FUNCTION FC 105 : VOID
VERSION : 0.1
VAR_TEMP
  Cmd_abbassa_indc : BOOL ;
  Cmd_alza_indc : BOOL ;
  Cmd_abbassa_indc_ibl : BOOL ;
  Cmd_alza_indc_ibl : BOOL ;
  Cmd_sblocca_pezzo : BOOL ;
  Cmd_blocca_pezzo : BOOL ;
  Cmd_sblocca_pezzo_ibl : BOOL ;
  Cmd_blocca_pezzo_ibl : BOOL ;
  Punt1 : DINT ;
  TempoTime : TIME ;
  TempoS5T : S5TIME ;
  Pos_comandata_asse_X : DINT ;
  Pos_comandata_asse_Y : DINT ;
  Tempo_ribaditura : DINT ;
END_VAR
BEGIN
NETWORK
TITLE = ******************       Diagnostica       *******************
NETWORK
TITLE = Allarmi di emergenza
NETWORK
TITLE = Controllo toolcode 
      L     DB106.DBB 0;
      L     W#16#1F;
      AW;
      L     DB110.DBW 36;
      <>I;
      AN    DB110.DBX 78.0;
//      S     "Op10.Bench.Alarms".Emegency.Alarm02
      S     DB104.DBX 9.1;
NETWORK
TITLE = Allarmi di STOP CICLO
NETWORK
TITLE = Controllo anelli adattamento
      A     DB110.DBX 38.0;
      AN    DB106.DBX 0.5;
      O(;
      AN    DB110.DBX 38.0;
      A     DB106.DBX 0.5;
      );
      AN    DB110.DBX 78.1;
      S     DB104.DBX 8.0;
      A     DB110.DBX 38.1;
      AN    DB106.DBX 0.6;
      O(;
      AN    DB110.DBX 38.1;
      A     DB106.DBX 0.6;
      );
      AN    DB110.DBX 78.1;
      S     DB104.DBX 8.1;
NETWORK
TITLE = Allarmi di NON START CICLO
NETWORK
TITLE = Allarmi di Warning
NETWORK
TITLE = Diagnostica: Hold Macchina
      AN    DB100.DBX 2.0;
      A(;
      A     DB100.DBX 0.4;
      AN    DB100.DBX 2.1;
      A     DB105.DBX 10.1;
      O(;
      A     DB100.DBX 0.3;
      A     DB105.DBX 10.0;
      );
      );
      =     DB100.DBX 2.4;
NETWORK
TITLE = ******************          Stati            *******************
      A     DB101.DBX 0.1;
      =     DB105.DBX 10.3;
      A     DB101.DBX 0.2;
      =     DB105.DBX 10.2;
NETWORK
TITLE =
      A     DB55.DBX 10.4;
      =     DB105.DBX 11.3;
      A     DB55.DBX 10.3;
      =     DB105.DBX 11.4;
      A     DB55.DBX 10.2;
      =     DB105.DBX 11.5;
      AN    DB55.DBX 11.2;
      AN    DB55.DBX 12.2;
      =     DB105.DBX 12.4;
NETWORK
TITLE = Stato: Fronte Start Ciclo
      A     DB101.DBX 0.0;
      FP    M 50.2;
      =     DB105.DBX 0.6;
NETWORK
TITLE = Lampade
      A     DB105.DBX 12.2;
      A     DB100.DBX 0.4;
      O     DB105.DBX 0.1;
      =     DB102.DBX 0.0;
      A     DB105.DBX 12.3;
      A     DB100.DBX 0.4;
      O     DB105.DBX 0.1;
      =     DB102.DBX 0.1;
NETWORK
TITLE = Cycle Type
NETWORK
TITLE = ******************         Sistemi           *******************
NETWORK
TITLE = Alza/abbassa Index cassetto
//*************************** COMANDI DA CICLI *************************
      A     DB120.DBX 9.5;
      O     DB120.DBX 12.3;
      O     DB120.DBX 31.7;
      =     DB105.DBX 0.2;
      A     DB120.DBX 10.0;
      A     DB105.DBX 10.2;
      O(;
      A     DB120.DBX 13.0;
      O     DB120.DBX 32.4;
      A     DB105.DBX 10.3;
      );
      =     DB105.DBX 0.3;
//*************************** COMANDI SENZA INTERBLOCCHI ***************
//CMD---------->Comando abbassa index cassetto
//MANUALE
      A     DB70.DBX 12.4;
      A     DB51.DBX 2.3;
      A     DB100.DBX 0.3;
//AUTOMATICO
      O(;
      A     DB100.DBX 0.4;
      AN    DB100.DBX 2.6;
      A     DB105.DBX 0.2;
      );
//SICUREZZA
      A     DB100.DBX 2.4;
      =     #Cmd_abbassa_indc;
//CMD---------->Comando alza index cassetto
//MANUALE
      A     DB70.DBX 12.4;
      A     DB51.DBX 2.2;
      A     DB100.DBX 0.3;
//AUTOMATICO
      O(;
      A     DB100.DBX 0.4;
      AN    DB100.DBX 2.6;
      A     DB105.DBX 0.3;
      );
//SICUREZZA
      A     DB100.DBX 2.4;
      =     #Cmd_alza_indc;
//************************** INTERBLOCCHI (E SEGNALAZIONE) ****************************
      A     DB105.DBX 0.0;
      O     DB105.DBX 10.2;
      O     DB105.DBX 10.3;
      R     DB104.DBX 24.0;
      A     #Cmd_alza_indc;
      A(;
      AN    DB105.DBX 10.2;
      AN    DB105.DBX 10.3;
      );
      S     DB104.DBX 24.0;
// MSG sblocco solo con ribaditrice alta
      A     DB105.DBX 0.0;
      O     DB105.DBX 11.3;
      R     DB104.DBX 24.2;
      A     #Cmd_abbassa_indc;
      AN    DB105.DBX 11.3;
      S     DB104.DBX 24.2;
// MSG sblocco solo con assi fermi
      A     DB105.DBX 0.0;
      O     DB105.DBX 12.4;
      R     DB104.DBX 24.3;
      A     #Cmd_abbassa_indc;
      AN    DB105.DBX 12.4;
      S     DB104.DBX 24.3;
// MSG sblocco solo con pezzo bloccato
      A     DB105.DBX 0.0;
      O     DB105.DBX 10.6;
      R     DB104.DBX 24.4;
      A     #Cmd_abbassa_indc;
      AN    DB105.DBX 10.6;
      S     DB104.DBX 24.4;
//************************** COMANDI CON INTERBLOCCHI ******************************
      AN    DB104.DBX 24.2;
      AN    DB104.DBX 24.3;
      AN    DB104.DBX 24.4;
      A     #Cmd_abbassa_indc;
      =     #Cmd_abbassa_indc_ibl;
      AN    DB104.DBX 24.0;
      A     #Cmd_alza_indc;
      =     #Cmd_alza_indc_ibl;
      CALL  FB 102 , DB 401 (
           DIX 0.0                  := TRUE,
           DIX 0.1                  := #Cmd_alza_indc_ibl,
           DIX 0.2                  := #Cmd_abbassa_indc_ibl,
           DIX 0.3                  := DB101.DBX 0.4,
           DIX 0.4                  := DB101.DBX 0.3,
           DIX 0.5                  := DB105.DBX 0.0,
           DID 2                    := L#2000,
           DIX 6.0                  := FALSE,
           DIX 8.0                  := DB102.DBX 0.3,
           DIX 8.1                  := DB102.DBX 0.2,
           DIX 8.2                  := DB105.DBX 10.5,
           DIX 8.3                  := DB105.DBX 10.4,
           DIX 8.4                  := DB104.DBX 8.2,
           DIX 8.5                  := DB104.DBX 8.3,
           DIX 8.6                  := DB104.DBX 8.4);
NETWORK
TITLE = Blocco/Sblocco pezzo
//*************************** COMANDI DA CICLI *************************
      A     DB120.DBX 13.0;
      O     DB120.DBX 32.4;
      A     DB101.DBX 0.4;
      A     DB105.DBX 10.3;
      =     DB105.DBX 0.4;
      A     DB120.DBX 9.5;
      O     DB120.DBX 10.0;
      =     DB105.DBX 0.5;
//*************************** COMANDI SENZA INTERBLOCCHI ***************
//CMD---------->Comando sblocco
//MANUALE
      A     DB70.DBX 12.5;
      A     DB51.DBX 2.2;
      A     DB100.DBX 0.3;
//AUTOMATICO
      O(;
      A     DB100.DBX 0.4;
      AN    DB100.DBX 2.6;
      A     DB105.DBX 0.4;
      );
//SICUREZZA
      A     DB100.DBX 2.4;
      =     #Cmd_sblocca_pezzo;
//CMD---------->Comando alza ribaditrice
//MANUALE
      A     DB70.DBX 12.5;
      A     DB51.DBX 2.3;
      A     DB100.DBX 0.3;
//AUTOMATICO
      O(;
      A     DB100.DBX 0.4;
      AN    DB100.DBX 2.6;
      A     DB105.DBX 0.5;
      );
//SICUREZZA
      A     DB100.DBX 2.4;
      =     #Cmd_blocca_pezzo;
//************************** INTERBLOCCHI (E SEGNALAZIONE) ****************************
//MSG---> Segnalazione interblocco Movimento ribaditrice non ammesso con motore ribaditrice in marcia
      A     DB105.DBX 0.0;
      O(;
      A     DB105.DBX 10.3;
      A     DB105.DBX 10.5;
      );
      R     DB104.DBX 24.1;
      A     #Cmd_sblocca_pezzo;
      A(;
      AN    DB105.DBX 10.3;
      ON    DB105.DBX 10.5;
      );
      S     DB104.DBX 24.1;
//************************** COMANDI CON INTERBLOCCHI ******************************
//CMD-------------> Comando abbassa e alza
      AN    DB104.DBX 24.1;
      A     #Cmd_sblocca_pezzo;
      =     #Cmd_sblocca_pezzo_ibl;
      A     #Cmd_blocca_pezzo;
      =     #Cmd_blocca_pezzo_ibl;
      CALL  FB 102 , DB 402 (
           DIX 0.0                  := TRUE,
           DIX 0.1                  := #Cmd_sblocca_pezzo_ibl,
           DIX 0.2                  := #Cmd_blocca_pezzo_ibl,
           DIX 0.3                  := DB101.DBX 0.6,
           DIX 0.4                  := DB101.DBX 0.5,
           DIX 0.5                  := DB105.DBX 0.0,
           DID 2                    := L#4000,
           DIX 6.0                  := FALSE,
           DIX 8.0                  := DB102.DBX 0.4,
           DIX 8.1                  := DB102.DBX 0.5,
           DIX 8.2                  := DB105.DBX 10.7,
           DIX 8.3                  := DB105.DBX 10.6,
           DIX 8.4                  := DB104.DBX 8.5,
           DIX 8.5                  := DB104.DBX 8.6,
           DIX 8.6                  := DB104.DBX 8.7);
NETWORK
TITLE = Gestione numero ribaditura in corso
      AN    DB120.DBX 18.0;
      O     DB120.DBX 9.2;
      O     DB120.DBX 10.0;
      O     DB120.DBX 13.0;
      JCN   nAzz;
      L     0;
      T     DB105.DBW 20;
nAzz: NOP   0;
      A     DB120.DBX 10.4;
      FP    M 50.3;
      =     DB105.DBX 11.6;
      AN    DB105.DBX 11.6;
      JC    nIn;
      L     DB105.DBW 20;
      L     1;
      +I;
      T     DB105.DBW 20;
nIn:  NOP   0;
NETWORK
TITLE = Valori posizione ribaditura corrente
      L     DB105.DBW 20;
      L     0;
      >I;
      JC    Cal;
// Punto inesistente
      L     L#0;
      T     DB105.DBD 22;
      T     DB105.DBD 26;
      T     DB105.DBD 30;
      JU    Cen;
Cal:  NOP   0;	// Estrazione dati punto da ricetta
      L     DB105.DBW 20;
      L     1;
      -I;
      ITD;
      L     L#12;
      *D;
      L     L#82;
      +D;
      SLW   3;
      T     #Punt1;
      OPN   DB 110;
      L     DBD [#Punt1];
      T     #Pos_comandata_asse_X;
      L     #Punt1;
      L     32;
      +D;
      T     #Punt1;
      L     DBD [#Punt1];
      T     #Pos_comandata_asse_Y;
      L     #Punt1;
      L     32;
      +D;
      T     #Punt1;
      L     DBD [#Punt1];
      T     #Tempo_ribaditura;
      L     #Pos_comandata_asse_X;
      T     DB105.DBD 22;
      L     #Pos_comandata_asse_Y;
      T     DB105.DBD 26;
      L     #Tempo_ribaditura;
      T     DB105.DBD 30;
Cen:  NOP   0;
NETWORK
TITLE = Impegno, comandi e stati ribaditrice per lavoro su OP10
      A     DB120.DBX 10.0;
      O     DB120.DBX 10.4;
      O     DB120.DBX 11.1;
      O     DB120.DBX 11.6;
      A     DB120.DBX 18.0;
      O(;
      A     DB120.DBX 31.2;
      A     DB120.DBX 40.0;
      );
      =     DB105.DBX 0.7;
      A     DB120.DBX 10.4;
      O     DB120.DBX 11.1;
      O     DB120.DBX 11.6;
      =     DB105.DBX 1.1;
      A     DB120.DBX 11.1;
      A     DB105.DBX 11.0;
      =     DB105.DBX 1.2;
      A     DB120.DBX 9.5;
      AN    DB105.DBX 11.7;
      O     DB120.DBX 11.6;
      O     DB120.DBX 31.2;
      A     DB105.DBX 11.0;
      =     DB105.DBX 1.3;
      A     DB55.DBX 13.0;
      =     DB105.DBX 11.0;
NETWORK
TITLE = Ribaditura
      L     DB105.DBD 30;
      T     #TempoTime;
      CALL  FC 40 (
           $1                       := #TempoTime,
           $2                       := #TempoS5T);
      A     DB120.DBX 11.1;
      A     DB105.DBX 11.5;
      A     DB105.DBX 11.4;
      L     #TempoS5T;
      SD    T 10;
      A     T 10;
      =     DB105.DBX 11.2;
NETWORK
TITLE = Assi - movimenti per lavorazioni OP10
      A     DB120.DBX 10.4;
      A     DB55.DBX 13.0;
      =     DB105.DBX 1.0;
      A     DB55.DBX 11.1;
      A     DB55.DBX 12.1;
      A     DB55.DBX 13.0;
      =     DB105.DBX 11.1;
NETWORK
TITLE = Definizione pezzo buono o scarto
      A     DB120.DBX 12.3;
      S     DB105.DBX 12.2;
      A     DB101.DBX 0.6;
      R     DB105.DBX 12.2;
      A     DB120.DBX 40.0;
      A     DB106.DBX 0.7;
      AN    DB105.DBX 12.2;
      S     DB105.DBX 12.3;
      A     DB101.DBX 0.6;
      R     DB105.DBX 12.3;
END_FUNCTION

FUNCTION FC 106 : VOID
VERSION : 0.1
VAR_INPUT
  ToolType : INT ;
END_VAR
VAR_OUTPUT
  ErrorToolType : BOOL ;
END_VAR
BEGIN
NETWORK
TITLE = Tool 1 - mappa ingressi
// Definizione ingressi E3.0 - E4.6
      L     #ToolType;
      L     1;
      <>I;
      JC    no1;
      SET;
      R     #ErrorToolType;
// Tool 1 - mappa ingressi
      A     I 4.1;
      =     DB106.DBX 0.0;
      A     I 4.2;
      =     DB106.DBX 0.1;
      A     I 4.3;
      =     DB106.DBX 0.2;
      A     I 4.4;
      =     DB106.DBX 0.3;
      A     I 4.5;
      =     DB106.DBX 0.4;
      A     I 4.0;
      =     DB106.DBX 0.5;
      A     I 3.7;
      =     DB106.DBX 0.6;
      A     I 3.6;
      =     DB106.DBX 0.7;
      A     I 3.1;
      =     DB106.DBX 1.0;
      A     I 3.0;
      =     DB106.DBX 1.1;
      A     I 3.3;
      =     DB106.DBX 1.2;
      A     I 3.2;
      =     DB106.DBX 1.3;
      A     I 3.5;
      =     DB106.DBX 1.4;
      A     I 3.4;
      =     DB106.DBX 1.5;
      BEU;
no1:  NOP   0;
NETWORK
TITLE = Tool 2 - mappa ingressi
      L     #ToolType;
      L     2;
      <>I;
      JC    no2;
      SET;
      S     #ErrorToolType;
// Tool 2 - predisposto ma inesistente
      BEU;
no2:  NOP   0;
NETWORK
TITLE = Error Tool Type
      SET;
      S     #ErrorToolType;
END_FUNCTION

FUNCTION FC 120 : VOID
VERSION : 0.1
BEGIN
NETWORK
TITLE =
      A     DB100.DBX 0.4;
      FP    M 50.4;
      =     DB105.DBX 12.0;
      AN    DB100.DBX 2.1;
      AN    DB100.DBX 2.0;
      FP    M 50.5;
      =     DB105.DBX 12.1;
NETWORK
TITLE =
      A     DB105.DBX 12.0;
      O     DB105.DBX 12.1;
      A(;
      AN    DB105.DBX 10.3;
      ON    DB101.DBX 0.4;
      ON    DB101.DBX 0.6;
      );
      S     DB120.DBX 40.0;
      AN    DB100.DBX 0.4;
//      U     "OP10".Diagnostic.Alarm_Stop_Cycle
      O     DB100.DBX 2.0;
      O     DB101.DBX 0.7;
      O     DB120.DBX 37.4;
      R     DB120.DBX 40.0;
      CLR;
      =     DB100.DBX 2.6;
      CALL  FB 121 , DB 431 (
           DIX 0.0                  := DB120.DBX 40.0,
           DIX 0.1                  := DB100.DBX 2.6,
           DIX 0.2                  := FALSE,
           DIX 2.0                  := DB120.DBX 28.0,
           DIX 2.1                  := DB120.DBX 28.1,
           DIX 2.2                  := DB120.DBX 28.2,
           DIW 4                    := DB120.DBW 22,
           DIW 6                    := DB120.DBW 24,
           DIW 8                    := DB120.DBW 26);
NETWORK
TITLE =
      A     DB100.DBX 0.4;
      AN    DB100.DBX 2.1;
      AN    DB100.DBX 2.0;
      AN    DB120.DBX 40.0;
// condizione di sicurezza
      AN    DB101.DBX 0.7;
      =     DB120.DBX 18.0;
      CALL  FB 120 , DB 430 (
           DIX 0.0                  := DB120.DBX 18.0,
           DIX 0.1                  := DB100.DBX 2.6,
           DIX 0.2                  := FALSE,
           DIX 2.0                  := DB120.DBX 6.0,
           DIX 2.1                  := DB120.DBX 6.1,
           DIX 2.2                  := DB120.DBX 6.2,
           DIW 4                    := DB120.DBW 0,
           DIW 6                    := DB120.DBW 2,
           DIW 8                    := DB120.DBW 4);
END_FUNCTION

FUNCTION FC 150 : VOID
VERSION : 0.1
VAR_TEMP
  ErrorToolType : BOOL ;
END_VAR
BEGIN
NETWORK
TITLE =
NETWORK
TITLE =
      CALL  FC 151;
      CALL  FC 156 (
           ToolType                 := DB160.DBW 22,
           ErrorToolType            := #ErrorToolType);
      A     #ErrorToolType;
      A     DB160.DBX 50.0;
//      S     DB154.DBX    0.0
      S     DB154.DBX 8.6;
      CALL  FC 153;
NETWORK
TITLE =
      A     DB55.DBX 0.0;
      =     DB155.DBX 0.0;
      A     DB55.DBX 0.1;
      =     DB155.DBX 0.1;
      A     DB55.DBX 10.1;
      =     DB155.DBX 10.0;
      A     DB55.DBX 10.5;
      =     DB155.DBX 10.1;
      CALL  FC 21 (
           NumDBallarmi             := DB 154,
           Reset_Allarmi            := DB155.DBX 0.0,
           AllarmeEmergenza         := DB150.DBX 2.0,
           AllarmeStopCiclo         := DB150.DBX 2.1,
           AllarmeStartCiclo        := DB150.DBX 2.2,
           AllarmeWarning           := DB150.DBX 2.3);
// Bench mode = Line mode...
      A     DB50.DBX 0.0;
      =     DB150.DBX 0.0;
      A     DB50.DBX 0.1;
      =     DB150.DBX 0.1;
      A     DB50.DBX 0.2;
      =     DB150.DBX 0.2;
      A     DB50.DBX 0.3;
      =     DB150.DBX 0.3;
      A     DB50.DBX 0.4;
      =     DB150.DBX 0.4;
NETWORK
TITLE =
      CALL  FC 155;
      CALL  FC 170;
NETWORK
TITLE =
      CALL  FC 152;
END_FUNCTION

FUNCTION FC 151 : VOID
VERSION : 0.1
VAR_TEMP
  RetVal : WORD ;
  Tastatore : REAL ;
END_VAR
BEGIN
NETWORK
TITLE =
      A     I 10.4;
      =     DB151.DBX 0.2;
      A     I 10.6;
      =     DB151.DBX 0.3;
      A     I 10.5;
      =     DB151.DBX 0.4;
      A     I 10.3;
      =     DB151.DBX 0.5;
      A     I 10.2;
      =     DB151.DBX 0.6;
      A     I 10.1;
      =     DB151.DBX 0.7;
      A     I 10.0;
      =     DB151.DBX 1.0;
NETWORK
TITLE =
      CALL  FC 5 (
           $1                       := P#P 256.0,
           $2                       := L#1088421888,
           $3                       := L#0,
           $4                       := FALSE,
           $5                       := #RetVal,
           $6                       := #Tastatore);
      L     #Tastatore;
      L     DB153.DBD 0;
      -R;
      T     DB151.DBD 6;
END_FUNCTION

FUNCTION FC 152 : VOID
VERSION : 0.1
BEGIN
NETWORK
TITLE =
      A     DB152.DBX 0.0;
      =     Q 0.5;
      A     DB152.DBX 0.1;
      =     Q 0.6;
      A     DB152.DBX 0.2;
      =     Q 2.0;
      A     DB152.DBX 0.3;
      =     Q 2.1;
      A     DB152.DBX 0.4;
      =     Q 1.5;
      A     DB152.DBX 0.5;
      =     Q 1.6;
      A     DB152.DBX 0.6;
      =     Q 1.3;
      A     DB152.DBX 0.7;
      =     Q 1.4;
END_FUNCTION

FUNCTION FC 153 : VOID
VERSION : 0.1
BEGIN
NETWORK
TITLE =
// Impostato da pagina di configurazione su PO
//      L     3.808000e+000
//      T     "Op20.Bench.Config".Offset_Tastatore
END_FUNCTION

FUNCTION FC 155 : VOID
VERSION : 0.1
VAR_TEMP
  Cmd_abbassa_indc : BOOL ;
  Cmd_alza_indc : BOOL ;
  Cmd_abbassa_indc_ibl : BOOL ;
  Cmd_alza_indc_ibl : BOOL ;
  Cmd_sblocca_pezzo : BOOL ;
  Cmd_blocca_pezzo : BOOL ;
  Cmd_sblocca_pezzo_ibl : BOOL ;
  Cmd_blocca_pezzo_ibl : BOOL ;
  Cmd_AlzaGrPiant : BOOL ;
  Cmd_AbbassaGrPiant : BOOL ;
  Cmd_AlzaGrPiant_ibl : BOOL ;
  Cmd_AbbassaGrPiant_ibl : BOOL ;
  Cmd_AlzaPiant : BOOL ;
  Cmd_AbbassaPiant : BOOL ;
  Cmd_AlzaPiant_ibl : BOOL ;
  Cmd_AbbassaPiant_ibl : BOOL ;
  CorsaMinRaggiunta : BOOL ;
  CorsaMaxSuperata : BOOL ;
  TempoTime : TIME ;
  TempoS5T : S5TIME ;
END_VAR
BEGIN
NETWORK
TITLE = ******************       Diagnostica       *******************
NETWORK
TITLE = Allarmi di emergenza
NETWORK
TITLE = Controllo toolcode 
      L     DB156.DBB 0;
      L     W#16#1F;
      AW;
      L     DB160.DBW 24;
      <>I;
      A     DB160.DBX 50.0;
//      S     "Op20.Bench.Alarms".Emegency.Alarm02
      S     DB154.DBX 8.7;
NETWORK
TITLE = Allarmi di STOP CICLO
NETWORK
TITLE = Allarmi di NON START CICLO
NETWORK
TITLE = Allarmi di Warning
NETWORK
TITLE = Diagnostica: Hold Macchina
      AN    DB150.DBX 2.0;
      A(;
      A     DB150.DBX 0.4;
      AN    DB150.DBX 2.1;
      A     DB155.DBX 10.1;
      O(;
      A     DB150.DBX 0.3;
      A     DB155.DBX 10.0;
      );
      );
      =     DB150.DBX 2.4;
NETWORK
TITLE = ******************          Stati            *******************
      AN    DB151.DBX 0.2;
      =     DB155.DBX 10.3;
      A     DB151.DBX 0.2;
      =     DB155.DBX 10.2;
NETWORK
TITLE = Stato: Fronte Start Ciclo
NETWORK
TITLE = Lampade
      A     DB155.DBX 11.3;
      A     DB150.DBX 0.4;
      O     DB155.DBX 0.1;
      =     DB152.DBX 0.0;
      A     DB155.DBX 11.4;
      A     DB150.DBX 0.4;
      O     DB155.DBX 0.1;
      =     DB152.DBX 0.1;
NETWORK
TITLE = Cycle Type
NETWORK
TITLE = ******************         Sistemi           *******************
NETWORK
TITLE = Alza/abbassa Index cassetto
//*************************** COMANDI DA CICLI *************************
      A     DB170.DBX 12.3;
      O     DB170.DBX 31.7;
      =     DB155.DBX 0.2;
      A     DB170.DBX 9.7;
      =     DB155.DBX 0.3;
//*************************** COMANDI SENZA INTERBLOCCHI ***************
//CMD---------->Comando abbassa index cassetto
//MANUALE
      A     DB70.DBX 12.6;
      A     DB51.DBX 2.3;
      A     DB150.DBX 0.3;
//AUTOMATICO
      O(;
      A     DB150.DBX 0.4;
      AN    DB150.DBX 2.6;
      A     DB155.DBX 0.2;
      );
//SICUREZZA
      A     DB150.DBX 2.4;
      =     #Cmd_abbassa_indc;
//CMD---------->Comando alza index cassetto
//MANUALE
      A     DB70.DBX 12.6;
      A     DB51.DBX 2.2;
      A     DB150.DBX 0.3;
//AUTOMATICO
      O(;
      A     DB150.DBX 0.4;
      AN    DB150.DBX 2.6;
      A     DB155.DBX 0.3;
      );
//SICUREZZA
      A     DB150.DBX 2.4;
      =     #Cmd_alza_indc;
//************************** INTERBLOCCHI (E SEGNALAZIONE) ****************************
      A     DB155.DBX 0.0;
      O     DB155.DBX 10.2;
      O     DB155.DBX 10.3;
      R     DB154.DBX 24.0;
      A     #Cmd_alza_indc;
      AN    DB155.DBX 10.2;
      S     DB154.DBX 24.0;
// Msg 
      A     DB155.DBX 0.0;
      O(;
      A     DB155.DBX 10.6;
      A     DB155.DBX 11.0;
      );
      R     DB154.DBX 24.4;
      AN    DB155.DBX 10.6;
      ON    DB155.DBX 11.0;
      A     #Cmd_abbassa_indc;
      S     DB154.DBX 24.4;
//************************** COMANDI CON INTERBLOCCHI ******************************
      AN    DB154.DBX 24.4;
      A     #Cmd_abbassa_indc;
      =     #Cmd_abbassa_indc_ibl;
      AN    DB154.DBX 24.0;
      A     #Cmd_alza_indc;
      =     #Cmd_alza_indc_ibl;
      CALL  FB 102 , DB 403 (
           DIX 0.0                  := TRUE,
           DIX 0.1                  := #Cmd_alza_indc_ibl,
           DIX 0.2                  := #Cmd_abbassa_indc_ibl,
           DIX 0.3                  := DB151.DBX 0.4,
           DIX 0.4                  := DB151.DBX 0.3,
           DIX 0.5                  := DB155.DBX 0.0,
           DID 2                    := L#1500,
           DIX 6.0                  := FALSE,
           DIX 8.0                  := DB152.DBX 0.3,
           DIX 8.1                  := DB152.DBX 0.2,
           DIX 8.2                  := DB155.DBX 10.5,
           DIX 8.3                  := DB155.DBX 10.4,
           DIX 8.4                  := DB154.DBX 8.1,
           DIX 8.5                  := DB154.DBX 8.2,
           DIX 8.6                  := DB154.DBX 8.3);
NETWORK
TITLE = Alza/abbassa gruppo di piantaggio
//*************************** COMANDI DA CICLI *************************
      A     DB170.DBX 11.6;
      O     DB170.DBX 31.2;
      A     DB155.DBX 11.0;
      =     DB155.DBX 0.4;
      A     DB170.DBX 10.4;
      =     DB155.DBX 0.5;
//*************************** COMANDI SENZA INTERBLOCCHI ***************
//CMD---------->Comando alza gruppo
//MANUALE
      A     DB70.DBX 12.7;
      A     DB51.DBX 2.3;
      A     DB150.DBX 0.3;
//AUTOMATICO
      O(;
      A     DB150.DBX 0.4;
      AN    DB150.DBX 2.6;
      A     DB155.DBX 0.4;
      );
//SICUREZZA
//      U     "OP20".Diagnostic.Safe_State
      A     DB155.DBX 10.0;
      =     #Cmd_AlzaGrPiant;
//CMD---------->Comando abbassa gruppo
//MANUALE
      A     DB70.DBX 12.7;
      A     DB51.DBX 2.2;
      A     DB150.DBX 0.3;
//AUTOMATICO
      O(;
      A     DB150.DBX 0.4;
      AN    DB150.DBX 2.6;
      A     DB155.DBX 0.5;
      );
//SICUREZZA
      A     DB150.DBX 2.4;
      =     #Cmd_AbbassaGrPiant;
//************************** INTERBLOCCHI (E SEGNALAZIONE) ****************************
      A     DB155.DBX 0.0;
      O     DB155.DBX 10.2;
      R     DB154.DBX 24.5;
      A     #Cmd_AbbassaGrPiant;
      AN    DB155.DBX 10.2;
      S     DB154.DBX 24.5;
      A     DB155.DBX 0.0;
      O     DB155.DBX 10.5;
      R     DB154.DBX 24.6;
      A     #Cmd_AbbassaGrPiant;
      AN    DB155.DBX 10.5;
      S     DB154.DBX 24.6;
      A     DB155.DBX 0.0;
      O     DB155.DBX 11.0;
      R     DB154.DBX 25.0;
      A     #Cmd_AlzaGrPiant;
      AN    DB155.DBX 11.0;
      S     DB154.DBX 25.0;
//************************** COMANDI CON INTERBLOCCHI ******************************
      AN    DB154.DBX 25.0;
      A     #Cmd_AlzaGrPiant;
      =     #Cmd_AlzaGrPiant_ibl;
      AN    DB154.DBX 24.5;
      AN    DB154.DBX 24.6;
      A     #Cmd_AbbassaGrPiant;
      =     #Cmd_AbbassaGrPiant_ibl;
      CALL  FB 102 , DB 404 (
           DIX 0.0                  := TRUE,
           DIX 0.1                  := #Cmd_AbbassaGrPiant_ibl,
           DIX 0.2                  := #Cmd_AlzaGrPiant_ibl,
           DIX 0.3                  := DB151.DBX 0.7,
           DIX 0.4                  := DB151.DBX 1.0,
           DIX 0.5                  := DB155.DBX 0.0,
           DID 2                    := L#3000,
           DIX 6.0                  := FALSE,
           DIX 8.0                  := DB152.DBX 0.6,
           DIX 8.1                  := DB152.DBX 0.7,
           DIX 8.2                  := DB155.DBX 10.7,
           DIX 8.3                  := DB155.DBX 10.6,
           DIX 8.4                  := DB154.DBX 8.0,
           DIX 8.5                  := DB154.DBX 8.1,
           DIX 8.6                  := DB154.DBX 8.2);
NETWORK
TITLE = Alza/abbassa cilindro di piantaggio
//*************************** COMANDI DA CICLI *************************
      A     DB170.DBX 11.6;
      O     DB170.DBX 31.2;
      =     DB155.DBX 0.6;
      A     DB170.DBX 11.1;
      =     DB155.DBX 0.7;
//*************************** COMANDI SENZA INTERBLOCCHI ***************
//CMD---------->Comando alza gruppo
//MANUALE
      A     DB70.DBX 13.0;
      A     DB51.DBX 2.3;
      A     DB150.DBX 0.3;
//AUTOMATICO
      O(;
      A     DB150.DBX 0.4;
      AN    DB150.DBX 2.6;
      A     DB155.DBX 0.6;
      );
//SICUREZZA
      A     DB150.DBX 2.4;
      =     #Cmd_AlzaPiant;
//CMD---------->Comando abbassa gruppo
//MANUALE
      A     DB70.DBX 13.0;
      A     DB51.DBX 2.2;
      A     DB150.DBX 0.3;
//AUTOMATICO
      O(;
      A     DB150.DBX 0.4;
      AN    DB150.DBX 2.6;
      A     DB155.DBX 0.7;
      );
//SICUREZZA
      A     DB150.DBX 2.4;
      =     #Cmd_AbbassaPiant;
//************************** INTERBLOCCHI (E SEGNALAZIONE) ****************************
      A     #Cmd_AbbassaPiant;
      AN    DB155.DBX 10.2;
      S     DB154.DBX 24.5;
      A     #Cmd_AbbassaPiant;
      AN    DB155.DBX 10.5;
      S     DB154.DBX 24.6;
      A     DB155.DBX 0.0;
      O     DB155.DBX 10.7;
      R     DB154.DBX 24.7;
      A     #Cmd_AbbassaPiant;
      AN    DB155.DBX 10.7;
      S     DB154.DBX 24.7;
//************************** COMANDI CON INTERBLOCCHI ******************************
      A     #Cmd_AlzaPiant;
      =     #Cmd_AlzaPiant_ibl;
      AN    DB154.DBX 24.5;
      AN    DB154.DBX 24.6;
      AN    DB154.DBX 24.7;
      A     #Cmd_AbbassaPiant;
      =     #Cmd_AbbassaPiant_ibl;
      CALL  FB 102 , DB 405 (
           DIX 0.0                  := TRUE,
           DIX 0.1                  := #Cmd_AbbassaPiant_ibl,
           DIX 0.2                  := #Cmd_AlzaPiant_ibl,
           DIX 0.3                  := DB151.DBX 0.5,
           DIX 0.4                  := DB151.DBX 0.6,
           DIX 0.5                  := DB155.DBX 0.0,
           DID 2                    := L#10000,
           DIX 6.0                  := FALSE,
           DIX 8.0                  := DB152.DBX 0.4,
           DIX 8.1                  := DB152.DBX 0.5,
           DIX 8.2                  := DB155.DBX 11.1,
           DIX 8.3                  := DB155.DBX 11.0,
           DIX 8.4                  := DB154.DBX 8.3,
           DIX 8.5                  := DB154.DBX 8.4,
           DIX 8.6                  := DB154.DBX 8.5);
NETWORK
TITLE = Pressatua: controllo ciclo e definizione pezzo OK/KO
      L     DB151.DBD 6;
      L     DB160.DBD 80;
      >=R;
      =     #CorsaMinRaggiunta;
      L     DB151.DBD 6;
      L     DB160.DBD 84;
      >=R;
      =     #CorsaMaxSuperata;
// gestione timeout piantaggio
      L     DB160.DBD 96;
      T     #TempoTime;
      CALL  FC 40 (
           $1                       := #TempoTime,
           $2                       := #TempoS5T);
      A     DB170.DBX 11.1;
      L     #TempoS5T;
      SD    T 21;
// Tempo di piantagio
      L     DB160.DBD 92;
      T     #TempoTime;
      CALL  FC 40 (
           $1                       := #TempoTime,
           $2                       := #TempoS5T);
      A     DB170.DBX 11.1;
      A     #CorsaMinRaggiunta;
      L     #TempoS5T;
      SD    T 22;
// definizione pezzo buono o scartgo
      A     T 21;
      O     #CorsaMaxSuperata;
      A     DB170.DBX 11.1;
      O     DB170.DBX 40.0;
      S     DB155.DBX 11.4;
      A     T 22;
      A     DB170.DBX 11.1;
      S     DB155.DBX 11.3;
      A     DB170.DBX 9.7;
      R     DB155.DBX 11.4;
      R     DB155.DBX 11.3;
// fine operazione di piantaggio
      A     T 22;
      O     T 21;
      A     DB170.DBX 11.1;
      =     DB155.DBX 11.2;
END_FUNCTION

FUNCTION FC 156 : VOID
VERSION : 0.1
VAR_INPUT
  ToolType : INT ;
END_VAR
VAR_OUTPUT
  ErrorToolType : BOOL ;
END_VAR
BEGIN
NETWORK
TITLE = Tool 1 - mappa ingressi
      L     #ToolType;
      L     1;
      <>I;
      JC    no1;
      SET;
      R     #ErrorToolType;
// Tool 1 - mappa ingressi
      A     I 2.3;
      =     DB156.DBX 0.0;
      A     I 2.4;
      =     DB156.DBX 0.1;
      A     I 2.5;
      =     DB156.DBX 0.2;
      A     I 2.6;
      =     DB156.DBX 0.3;
      A     I 2.7;
      =     DB156.DBX 0.4;
      BEU;
no1:  NOP   0;
NETWORK
TITLE = Tool 2 - mappa ingressi
      L     #ToolType;
      L     2;
      <>I;
      JC    no2;
      SET;
      S     #ErrorToolType;
// Tool 2 - predisposto ma inesistente
      BEU;
no2:  NOP   0;
NETWORK
TITLE = Error Tool Type
      SET;
      S     #ErrorToolType;
END_FUNCTION

FUNCTION FC 170 : VOID
VERSION : 0.1
BEGIN
NETWORK
TITLE =
      A     DB150.DBX 0.4;
      FP    M 51.6;
      =     DB155.DBX 11.5;
      AN    DB150.DBX 2.1;
      AN    DB150.DBX 2.0;
      FP    M 51.7;
      =     DB155.DBX 11.6;
NETWORK
TITLE =
      A     DB155.DBX 11.5;
      O     DB155.DBX 11.6;
      A(;
      AN    DB151.DBX 0.3;
      ON    DB151.DBX 1.0;
      ON    DB151.DBX 0.6;
      );
      S     DB170.DBX 40.0;
      AN    DB150.DBX 0.4;
      O     DB150.DBX 2.1;
      O     DB150.DBX 2.0;
      O     DB170.DBX 37.4;
      R     DB170.DBX 40.0;
      CLR;
      =     DB150.DBX 2.6;
      CALL  FB 171 , DB 437 (
           IN_Cm_ON                 := DB170.DBX 40.0,
           IN_HOLD                  := DB150.DBX 2.6,
           IN_STEP                  := FALSE,
           OUT_St_CicloInCorso      := DB170.DBX 28.0,
           OUT_St_CicloTerminatoOK  := DB170.DBX 28.1,
           OUT_St_CicloTerminatoKO  := DB170.DBX 28.2,
           OUT_CicloStato           := DB170.DBW 22,
           OUT_Page                 := DB170.DBW 24,
           OUT_Message              := DB170.DBW 26);
NETWORK
TITLE =
      A     DB150.DBX 0.4;
      AN    DB150.DBX 2.1;
      AN    DB150.DBX 2.0;
      AN    DB170.DBX 40.0;
// condizione di sicurezza
      =     DB170.DBX 18.0;
      CALL  FB 170 , DB 438 (
           IN_Cm_ON                 := DB170.DBX 18.0,
           IN_HOLD                  := DB150.DBX 2.6,
           IN_STEP                  := FALSE,
           OUT_St_CicloInCorso      := DB170.DBX 6.0,
           OUT_St_CicloTerminatoOK  := DB170.DBX 6.1,
           OUT_St_CicloTerminatoKO  := DB170.DBX 6.2,
           OUT_CicloStato           := DB170.DBW 0,
           OUT_Page                 := DB170.DBW 2,
           OUT_Message              := DB170.DBW 4);
END_FUNCTION

FUNCTION FC 200 : VOID
VERSION : 0.1
VAR_TEMP
  ErrorToolType : BOOL ;
END_VAR
BEGIN
NETWORK
TITLE =
NETWORK
TITLE =
      CALL  FC 201;
      CALL  FC 206 (
           ToolType                 := DB210.DBW 34,
           ErrorToolType            := #ErrorToolType);
      A     #ErrorToolType;
      AN    DB210.DBX 78.0;
//      S     DB204.DBX    0.0
      S     DB204.DBX 9.0;
      CALL  FC 203;
NETWORK
TITLE =
      A     DB55.DBX 0.0;
      =     DB205.DBX 0.0;
      A     DB55.DBX 0.1;
      =     DB205.DBX 0.1;
      A     DB55.DBX 10.1;
      =     DB205.DBX 10.0;
      A     DB55.DBX 10.5;
      =     DB205.DBX 10.1;
      CALL  FC 21 (
           NumDBallarmi             := DB 204,
           Reset_Allarmi            := DB205.DBX 0.0,
           AllarmeEmergenza         := DB200.DBX 2.0,
           AllarmeStopCiclo         := DB200.DBX 2.1,
           AllarmeStartCiclo        := DB200.DBX 2.2,
           AllarmeWarning           := DB200.DBX 2.3);
      A     DB50.DBX 0.0;
      =     DB200.DBX 0.0;
      A     DB50.DBX 0.1;
      =     DB200.DBX 0.1;
      A     DB50.DBX 0.2;
      =     DB200.DBX 0.2;
      A     DB50.DBX 0.3;
      =     DB200.DBX 0.3;
      A     DB50.DBX 0.4;
      =     DB200.DBX 0.4;
NETWORK
TITLE =
      CALL  FC 205;
      CALL  FC 220;
NETWORK
TITLE =
      CALL  FC 202;
END_FUNCTION

FUNCTION FC 201 : VOID
VERSION : 0.1
BEGIN
NETWORK
TITLE =
      A     I 6.1;
      =     DB201.DBX 0.0;
      A     I 9.6;
      =     DB201.DBX 0.1;
      AN    I 9.0;
      =     DB201.DBX 0.2;
      A     I 9.1;
      =     DB201.DBX 0.3;
      A     I 9.2;
      =     DB201.DBX 0.4;
      A     I 9.3;
      =     DB201.DBX 0.5;
      A     I 9.4;
      =     DB201.DBX 0.6;
      A     I 9.5;
      =     DB201.DBX 0.7;
      AN    I 1.5;
      =     DB201.DBX 1.0;
END_FUNCTION

FUNCTION FC 202 : VOID
VERSION : 0.1
BEGIN
NETWORK
TITLE =
      A     DB202.DBX 0.0;
      =     Q 0.1;
      A     DB202.DBX 0.1;
      =     Q 0.2;
      A     DB202.DBX 0.2;
      =     Q 2.6;
      A     DB202.DBX 0.3;
      =     Q 2.7;
      A     DB202.DBX 0.4;
      =     Q 3.1;
      A     DB202.DBX 0.5;
      =     Q 3.0;
END_FUNCTION

FUNCTION FC 203 : VOID
VERSION : 0.1
BEGIN
NETWORK
TITLE =
END_FUNCTION

FUNCTION FC 205 : VOID
VERSION : 0.1
VAR_TEMP
  Cmd_abbassa_indc : BOOL ;
  Cmd_alza_indc : BOOL ;
  Cmd_abbassa_indc_ibl : BOOL ;
  Cmd_alza_indc_ibl : BOOL ;
  Cmd_sblocca_pezzo : BOOL ;
  Cmd_blocca_pezzo : BOOL ;
  Cmd_sblocca_pezzo_ibl : BOOL ;
  Cmd_blocca_pezzo_ibl : BOOL ;
  Punt1 : DINT ;
  TempoTime : TIME ;
  TempoS5T : S5TIME ;
  Pos_comandata_asse_X : DINT ;
  Pos_comandata_asse_Y : DINT ;
  Tempo_ribaditura : DINT ;
END_VAR
BEGIN
NETWORK
TITLE = ******************       Diagnostica       *******************
NETWORK
TITLE = Allarmi di emergenza
NETWORK
TITLE = Controllo toolcode 
      L     DB206.DBB 0;
      L     W#16#1F;
      AW;
      L     DB210.DBW 36;
      <>I;
      AN    DB210.DBX 78.0;
//      S     DB204.DBX    0.1
      S     DB204.DBX 9.1;
NETWORK
TITLE = Allarmi di STOP CICLO
NETWORK
TITLE = Controllo anelli adattamento
      A     DB210.DBX 38.0;
      AN    DB206.DBX 0.5;
      O(;
      AN    DB210.DBX 38.0;
      A     DB206.DBX 0.5;
      );
      AN    DB210.DBX 78.1;
      S     DB204.DBX 8.0;
      A     DB210.DBX 38.1;
      AN    DB206.DBX 0.6;
      O(;
      AN    DB210.DBX 38.1;
      A     DB206.DBX 0.6;
      );
      AN    DB210.DBX 78.1;
      S     DB204.DBX 8.1;
NETWORK
TITLE = Allarmi di NON START CICLO
NETWORK
TITLE = Allarmi di Warning
NETWORK
TITLE = Diagnostica: Hold Macchina
      AN    DB200.DBX 2.0;
      A(;
      A     DB200.DBX 0.4;
      AN    DB200.DBX 2.1;
      A     DB205.DBX 10.1;
      O(;
      A     DB200.DBX 0.3;
      A     DB205.DBX 10.0;
      );
      );
      =     DB200.DBX 2.4;
NETWORK
TITLE = ******************          Stati            *******************
      A     DB201.DBX 0.2;
      =     DB205.DBX 10.3;
      A     DB201.DBX 0.3;
      =     DB205.DBX 10.2;
NETWORK
TITLE =
      A     DB55.DBX 10.4;
      =     DB205.DBX 11.3;
      A     DB55.DBX 10.3;
      =     DB205.DBX 11.4;
      A     DB55.DBX 10.2;
      =     DB205.DBX 11.5;
      AN    DB55.DBX 11.2;
      AN    DB55.DBX 12.2;
      =     DB205.DBX 12.4;
NETWORK
TITLE = Stato: Fronte Start Ciclo
      A     DB201.DBX 0.0;
      FP    M 50.7;
      =     DB205.DBX 0.6;
NETWORK
TITLE = Lampade
      A     DB205.DBX 12.2;
      A     DB200.DBX 0.4;
      O     DB205.DBX 0.1;
      =     DB202.DBX 0.0;
      A     DB205.DBX 12.3;
      A     DB200.DBX 0.4;
      O     DB205.DBX 0.1;
      =     DB202.DBX 0.1;
NETWORK
TITLE = Cycle Type
NETWORK
TITLE = ******************         Sistemi           *******************
NETWORK
TITLE = Alza/abbassa Index cassetto
//*************************** COMANDI DA CICLI *************************
      A     DB220.DBX 9.5;
      O     DB220.DBX 12.3;
      O     DB220.DBX 31.7;
      =     DB205.DBX 0.2;
      A     DB220.DBX 10.0;
      A     DB205.DBX 10.2;
      O(;
      A     DB220.DBX 13.0;
      O     DB220.DBX 32.4;
      A     DB205.DBX 10.3;
      );
      =     DB205.DBX 0.3;
//*************************** COMANDI SENZA INTERBLOCCHI ***************
//CMD---------->Comando abbassa index cassetto
//MANUALE
      A     DB70.DBX 13.1;
      A     DB51.DBX 2.3;
      A     DB200.DBX 0.3;
//AUTOMATICO
      O(;
      A     DB200.DBX 0.4;
      AN    DB200.DBX 2.6;
      A     DB205.DBX 0.2;
      );
//SICUREZZA
      A     DB200.DBX 2.4;
      =     #Cmd_abbassa_indc;
//CMD---------->Comando alza index cassetto
//MANUALE
      A     DB70.DBX 13.1;
      A     DB51.DBX 2.2;
      A     DB200.DBX 0.3;
//AUTOMATICO
      O(;
      A     DB200.DBX 0.4;
      AN    DB200.DBX 2.6;
      A     DB205.DBX 0.3;
      );
//SICUREZZA
      A     DB200.DBX 2.4;
      =     #Cmd_alza_indc;
//************************** INTERBLOCCHI (E SEGNALAZIONE) ****************************
      A     DB205.DBX 0.0;
      O     DB205.DBX 10.2;
      O     DB205.DBX 10.3;
      R     DB204.DBX 24.0;
      A     #Cmd_alza_indc;
      A(;
      AN    DB205.DBX 10.2;
      AN    DB205.DBX 10.3;
      );
      S     DB204.DBX 24.0;
// MSG sblocco solo con ribaditrice alta
      A     DB205.DBX 0.0;
      O     DB205.DBX 11.3;
      R     DB204.DBX 24.2;
      A     #Cmd_abbassa_indc;
      AN    DB205.DBX 11.3;
      S     DB204.DBX 24.2;
// MSG sblocco solo con assi fermi
      A     DB205.DBX 0.0;
      O     DB205.DBX 12.4;
      R     DB204.DBX 24.3;
      A     #Cmd_abbassa_indc;
      AN    DB205.DBX 12.4;
      S     DB204.DBX 24.3;
// MSG sblocco solo con pezzo bloccato
      A     DB205.DBX 0.0;
      O     DB205.DBX 10.7;
      R     DB204.DBX 24.4;
      A     #Cmd_abbassa_indc;
      AN    DB205.DBX 10.7;
      S     DB204.DBX 24.4;
//************************** COMANDI CON INTERBLOCCHI ******************************
      AN    DB204.DBX 24.2;
      AN    DB204.DBX 24.3;
      AN    DB204.DBX 24.4;
      A     #Cmd_abbassa_indc;
      =     #Cmd_abbassa_indc_ibl;
      AN    DB204.DBX 24.0;
      A     #Cmd_alza_indc;
      =     #Cmd_alza_indc_ibl;
      CALL  FB 102 , DB 406 (
           DIX 0.0                  := TRUE,
           DIX 0.1                  := #Cmd_alza_indc_ibl,
           DIX 0.2                  := #Cmd_abbassa_indc_ibl,
           DIX 0.3                  := DB201.DBX 0.5,
           DIX 0.4                  := DB201.DBX 0.4,
           DIX 0.5                  := DB205.DBX 0.0,
           DID 2                    := L#3000,
           DIX 6.0                  := FALSE,
           DIX 8.0                  := DB202.DBX 0.3,
           DIX 8.1                  := DB202.DBX 0.2,
           DIX 8.2                  := DB205.DBX 10.5,
           DIX 8.3                  := DB205.DBX 10.4,
           DIX 8.4                  := DB204.DBX 8.2,
           DIX 8.5                  := DB204.DBX 8.3,
           DIX 8.6                  := DB204.DBX 8.4);
NETWORK
TITLE = Blocco/Sblocco pezzo
//*************************** COMANDI DA CICLI *************************
      A     DB220.DBX 9.2;
      O     DB220.DBX 13.0;
      O     DB220.DBX 32.4;
      A     DB201.DBX 0.5;
      A     DB205.DBX 10.3;
      =     DB205.DBX 0.4;
      A     DB220.DBX 9.3;
      O     DB120.DBX 10.0;
      =     DB205.DBX 0.5;
//*************************** COMANDI SENZA INTERBLOCCHI ***************
//CMD---------->Comando sblocco
//MANUALE
      A     DB70.DBX 13.2;
      A     DB51.DBX 2.2;
      A     DB200.DBX 0.3;
//AUTOMATICO
      O(;
      A     DB200.DBX 0.4;
      AN    DB200.DBX 2.6;
      A     DB205.DBX 0.4;
      );
//SICUREZZA
      A     DB200.DBX 2.4;
      =     #Cmd_sblocca_pezzo;
//CMD---------->Comando alza ribaditrice
//MANUALE
      A     DB70.DBX 13.2;
      A     DB51.DBX 2.3;
      A     DB200.DBX 0.3;
//AUTOMATICO
      O(;
      A     DB200.DBX 0.4;
      AN    DB200.DBX 2.6;
      A     DB205.DBX 0.5;
      );
//SICUREZZA
      A     DB200.DBX 2.4;
      =     #Cmd_blocca_pezzo;
//************************** INTERBLOCCHI (E SEGNALAZIONE) ****************************
//MSG---> Segnalazione interblocco Movimento ribaditrice non ammesso con motore ribaditrice in marcia
      A     DB205.DBX 0.0;
      O(;
      A     DB205.DBX 10.3;
      A     DB205.DBX 10.5;
      );
      R     DB204.DBX 24.1;
      A     #Cmd_sblocca_pezzo;
      A(;
      AN    DB205.DBX 10.3;
      ON    DB205.DBX 10.5;
      );
      S     DB204.DBX 24.1;
//************************** COMANDI CON INTERBLOCCHI ******************************
//CMD-------------> Comando abbassa e alza
      AN    DB204.DBX 24.1;
      A     #Cmd_sblocca_pezzo;
      =     #Cmd_sblocca_pezzo_ibl;
      A     #Cmd_blocca_pezzo;
      =     #Cmd_blocca_pezzo_ibl;
      CALL  FB 102 , DB 407 (
           DIX 0.0                  := TRUE,
           DIX 0.1                  := #Cmd_sblocca_pezzo_ibl,
           DIX 0.2                  := #Cmd_blocca_pezzo_ibl,
           DIX 0.3                  := DB201.DBX 0.7,
           DIX 0.4                  := DB201.DBX 0.6,
           DIX 0.5                  := DB205.DBX 0.0,
           DID 2                    := L#3000,
           DIX 6.0                  := FALSE,
           DIX 8.0                  := DB202.DBX 0.4,
           DIX 8.1                  := DB202.DBX 0.5,
           DIX 8.2                  := DB205.DBX 10.6,
           DIX 8.3                  := DB205.DBX 10.7,
           DIX 8.4                  := DB204.DBX 8.5,
           DIX 8.5                  := DB204.DBX 8.6,
           DIX 8.6                  := DB204.DBX 8.7);
NETWORK
TITLE = Gestione numero ribaditura in corso
      AN    DB220.DBX 18.0;
      O     DB220.DBX 9.2;
      O     DB220.DBX 10.0;
      O     DB220.DBX 13.0;
      JCN   nAzz;
      L     0;
      T     DB205.DBW 20;
nAzz: NOP   0;
      A     DB220.DBX 10.4;
      FP    M 50.6;
      =     DB205.DBX 11.6;
      AN    DB205.DBX 11.6;
      JC    nIn;
      L     DB205.DBW 20;
      L     1;
      +I;
      T     DB205.DBW 20;
nIn:  NOP   0;
NETWORK
TITLE = Valori posizione ribaditura corrente
      L     DB205.DBW 20;
      L     0;
      >I;
      JC    Cal;
// Punto inesistente
      L     L#0;
      T     DB205.DBD 22;
      T     DB205.DBD 26;
      T     DB205.DBD 30;
      JU    Cen;
Cal:  NOP   0;	// Estrazione dati punto da ricetta
      L     DB205.DBW 20;
      DEC   1;
      ITD;
      L     L#12;
      *D;
      L     L#82;
      +D;
      SLW   3;
      T     #Punt1;
      OPN   DB 210;
      L     DBD [#Punt1];
      T     #Pos_comandata_asse_X;
      L     #Punt1;
      L     32;
      +D;
      T     #Punt1;
      L     DBD [#Punt1];
      T     #Pos_comandata_asse_Y;
      L     #Punt1;
      L     32;
      +D;
      T     #Punt1;
      L     DBD [#Punt1];
      T     #Tempo_ribaditura;
      L     #Pos_comandata_asse_X;
      T     DB205.DBD 22;
      L     #Pos_comandata_asse_Y;
      T     DB205.DBD 26;
      L     #Tempo_ribaditura;
      T     DB205.DBD 30;
Cen:  NOP   0;
NETWORK
TITLE = Impegno, comandi e stati ribaditrice per lavoro su OP10
      A     DB220.DBX 10.0;
      O     DB220.DBX 10.4;
      O     DB220.DBX 11.1;
      O     DB220.DBX 11.6;
      A     DB220.DBX 18.0;
      O(;
      A     DB220.DBX 31.2;
      A     DB220.DBX 40.0;
      );
      =     DB205.DBX 0.7;
      A     DB220.DBX 10.4;
      O     DB220.DBX 11.1;
      O     DB220.DBX 11.6;
      =     DB205.DBX 1.1;
      A     DB220.DBX 11.1;
      A     DB205.DBX 11.0;
      =     DB205.DBX 1.2;
      A     DB220.DBX 9.5;
      AN    DB205.DBX 11.7;
      O     DB220.DBX 11.6;
      O     DB220.DBX 31.2;
      A     DB205.DBX 11.0;
      =     DB205.DBX 1.3;
      A     DB55.DBX 13.1;
      =     DB205.DBX 11.0;
NETWORK
TITLE = Ribaditura
      L     DB205.DBD 30;
      T     #TempoTime;
      CALL  FC 40 (
           $1                       := #TempoTime,
           $2                       := #TempoS5T);
      A     DB220.DBX 11.1;
      A     DB205.DBX 11.5;
      A     DB205.DBX 11.4;
      L     #TempoS5T;
      SD    T 11;
      A     T 11;
      =     DB205.DBX 11.2;
NETWORK
TITLE = Assi - movimenti per lavorazioni OP10
      A     DB220.DBX 10.4;
      A     DB55.DBX 13.1;
      =     DB205.DBX 1.0;
      A     DB55.DBX 11.1;
      A     DB55.DBX 12.1;
      A     DB55.DBX 13.1;
      =     DB205.DBX 11.1;
NETWORK
TITLE = Definizione pezzo buono o scarto
      A     DB220.DBX 12.3;
      S     DB205.DBX 12.2;
      A     DB201.DBX 0.7;
      R     DB205.DBX 12.2;
      A     DB220.DBX 40.0;
      A     DB206.DBX 0.7;
      AN    DB205.DBX 12.2;
      S     DB205.DBX 12.3;
      A     DB201.DBX 0.7;
      R     DB205.DBX 12.3;
END_FUNCTION

FUNCTION FC 206 : VOID
VERSION : 0.1
VAR_INPUT
  ToolType : INT ;
END_VAR
VAR_OUTPUT
  ErrorToolType : BOOL ;
END_VAR
BEGIN
NETWORK
TITLE = Tool 1 - mappa ingressi
      L     #ToolType;
      L     1;
      <>I;
      JC    no1;
      SET;
      R     #ErrorToolType;
// Tool 1 - mappa ingressi
      A     I 7.0;
      =     DB206.DBX 0.0;
      A     I 7.1;
      =     DB206.DBX 0.1;
      A     I 7.2;
      =     DB206.DBX 0.2;
      A     I 7.3;
      =     DB206.DBX 0.3;
      A     I 7.4;
      =     DB206.DBX 0.4;
      A     I 5.1;
      =     DB206.DBX 0.5;
      A     I 5.2;
      =     DB206.DBX 0.6;
      A     I 5.0;
      =     DB206.DBX 0.7;
      BEU;
no1:  NOP   0;
NETWORK
TITLE = Tool 2 - mappa ingressi
      L     #ToolType;
      L     2;
      <>I;
      JC    no2;
      SET;
      S     #ErrorToolType;
// Tool 2 - predisposto ma inesistente
      BEU;
no2:  NOP   0;
NETWORK
TITLE = Error Tool Type
      SET;
      S     #ErrorToolType;
END_FUNCTION

FUNCTION FC 220 : VOID
VERSION : 0.1
BEGIN
NETWORK
TITLE =
      A     DB200.DBX 0.4;
      FP    M 51.0;
      =     DB205.DBX 12.0;
      AN    DB200.DBX 2.1;
      AN    DB200.DBX 2.0;
      FP    M 51.1;
      =     DB205.DBX 12.1;
NETWORK
TITLE =
      A     DB205.DBX 12.0;
      O     DB205.DBX 12.1;
      A(;
      AN    DB205.DBX 10.3;
      ON    DB201.DBX 0.5;
      ON    DB201.DBX 0.7;
      );
      S     DB220.DBX 40.0;
      AN    DB200.DBX 0.4;
      O     DB200.DBX 2.1;
      O     DB200.DBX 2.0;
      O     DB201.DBX 1.0;
      O     DB220.DBX 37.4;
      R     DB220.DBX 40.0;
      CLR;
      =     DB200.DBX 2.6;
      CALL  FB 221 , DB 435 (
           DIX 0.0                  := DB220.DBX 40.0,
           DIX 0.1                  := DB200.DBX 2.6,
           DIX 0.2                  := FALSE,
           DIX 2.0                  := DB220.DBX 28.0,
           DIX 2.1                  := DB220.DBX 28.1,
           DIX 2.2                  := DB220.DBX 28.2,
           DIW 4                    := DB220.DBW 22,
           DIW 6                    := DB220.DBW 24,
           DIW 8                    := DB220.DBW 26);
NETWORK
TITLE =
      A     DB200.DBX 0.4;
      AN    DB200.DBX 2.1;
      AN    DB200.DBX 2.0;
      AN    DB220.DBX 40.0;
// condizione di sicurezza
      AN    DB201.DBX 1.0;
      =     DB220.DBX 18.0;
      CALL  FB 220 , DB 436 (
           DIX 0.0                  := DB220.DBX 18.0,
           DIX 0.1                  := DB200.DBX 2.6,
           DIX 0.2                  := FALSE,
           DIX 2.0                  := DB220.DBX 6.0,
           DIX 2.1                  := DB220.DBX 6.1,
           DIX 2.2                  := DB220.DBX 6.2,
           DIW 4                    := DB220.DBW 0,
           DIW 6                    := DB220.DBW 2,
           DIW 8                    := DB220.DBW 4);
END_FUNCTION

DATA_BLOCK DB 50
VERSION : 0.1
UDT 250
BEGIN
END_DATA_BLOCK

DATA_BLOCK DB 51
VERSION : 0.1
  STRUCT
   Q_Ribaditrice : BOOL ;
   Q_protezione_uscite : BOOL ;
   Q_Protez_circ_emergena : BOOL ;	//161QF1
   Q_Automatici_230_V : BOOL ;	//162F1-162F2-162F3-162F4
   Aux_OK : BOOL ;
   Ripari_OK : BOOL ;
   Anomalia_Condizionatore : BOOL ;
   Sequenza_fasi_OK : BOOL ;
   PLC_OK : BOOL ;	//Feedback relè PLC ok
   Chiave_Blocc_Porta_SX : BOOL ;
   Chiave_Blocc_Porta_DX : BOOL ;
   P_TestLampade : BOOL ;
   P_StartCiclo : BOOL ;	//??? che fa ???
   P_StopCiclo : BOOL ;
   S_Manuale : BOOL ;
   S_Automatico : BOOL ;
   Q_Azionam_Asse_X : BOOL ;
   Q_Azionam_Asse_Y : BOOL ;
   Jog_piu : BOOL ;
   Jog_meno : BOOL ;
   P_reset_allarmi : BOOL ;
   Pressostato_aria : BOOL ;
   Ribaditrice_bassa : BOOL ;
   Ribaditrice_alta : BOOL ;
   Press_aria_dpoop_EMG : BOOL ;
   Extracorsa_X : BOOL ;
   Extracorsa_Y : BOOL ;
   Ris_33 : BOOL ;
   Ris_34 : BOOL ;
   Ris_35 : BOOL ;
   Ris_36 : BOOL ;
   Ris_37 : BOOL ;
  END_STRUCT ;	
BEGIN
   Q_Ribaditrice := TRUE;
   Q_protezione_uscite := TRUE;
   Q_Protez_circ_emergena := TRUE;
   Q_Automatici_230_V := TRUE;
   Aux_OK := TRUE;
   Ripari_OK := TRUE;
   Sequenza_fasi_OK := TRUE;
   PLC_OK := TRUE;
   Chiave_Blocc_Porta_SX := TRUE;
   Chiave_Blocc_Porta_DX := TRUE;
   S_Automatico := TRUE;
   Q_Azionam_Asse_X := TRUE;
   Q_Azionam_Asse_Y := TRUE;
   Pressostato_aria := TRUE;
   Ribaditrice_alta := TRUE;
   Press_aria_dpoop_EMG := TRUE;
END_DATA_BLOCK

DATA_BLOCK DB 52
VERSION : 0.1
  STRUCT
   PLC_OK : BOOL ;
   Valvola_generale_aria : BOOL ;	//TOLTO!!!
   Marcia_ribaditrice : BOOL ;
   EV_abbassa_ribaditrice : BOOL ;
   Spare_0_4 : BOOL ;
   Blocco_porta_SX : BOOL ;
   Blocco_porta_DX : BOOL ;
   Lampeggiante_allarmi : BOOL ;
   LampPorteChiuse : BOOL ;
  END_STRUCT ;	
BEGIN
   PLC_OK := TRUE;
   Blocco_porta_SX := TRUE;
   Blocco_porta_DX := TRUE;
   LampPorteChiuse := TRUE;
END_DATA_BLOCK

DATA_BLOCK DB 53
VERSION : 0.1
  STRUCT
   Vel_max_assi_auto : DINT ;	//
   Vel_max_assi_man : DINT ;
   Accel_assi_auto : DINT ;
   Accel_assi_man : DINT ;
   Offset_attrezzo_OP10_X : DINT ;	//
   Offset_attrezzo_OP10_Y : DINT ;
   Offset_attrezzo_OP40_X : DINT ;	//
   Offset_attrezzo_OP40_Y : DINT ;
  END_STRUCT ;	
BEGIN
   Vel_max_assi_auto := L#15000;
   Vel_max_assi_man := L#15000;
   Accel_assi_auto := L#100;
   Accel_assi_man := L#100;
   Offset_attrezzo_OP10_X := L#71501;
   Offset_attrezzo_OP10_Y := L#47116;
   Offset_attrezzo_OP40_X := L#371523;
   Offset_attrezzo_OP40_Y := L#47047;
END_DATA_BLOCK

DATA_BLOCK DB 54
VERSION : 0.1
  STRUCT
   Emegency : STRUCT
    Alarm01 : BOOL ;	//Q_protezione_uscite
    Alarm02 : BOOL ;	//Protez_circ_emergena
    Alarm03 : BOOL ;	//Sequenza_fasi_OK
    Alarm04 : BOOL ;	//Q_Azionam_Asse_X
    Alarm05 : BOOL ;	//Q_Azionam_Asse_Y
    Alarm06 : BOOL ;	//Manca aria
    Alarm07 : BOOL ;	//Valvola aria inceppata
    Alarm08 : BOOL ;	//Errore comunicazione con Azionamento asse X
    Alarm09 : BOOL ;	//Errore comunicazione con Azionamento asse Y
    Alarm10 : BOOL ;	//Errore comunicazione con CU Azionamento asse X
    Alarm11 : BOOL ;	//Errore comunicazione con CU Azionamento asse Y
    Alarm12 : BOOL ;	//Extracorsa asse X
    Alarm13 : BOOL ;	//Extracorsa asse Y
    Alarm14 : BOOL ;	//Errore Relè PLC OK
    Alarm15 : BOOL ;
    Alarm16 : BOOL ;
    Alarm17 : BOOL ;
    Alarm18 : BOOL ;
    Alarm19 : BOOL ;
    Alarm20 : BOOL ;
    Alarm21 : BOOL ;
    Alarm22 : BOOL ;
    Alarm23 : BOOL ;
    Alarm24 : BOOL ;
    Alarm25 : BOOL ;
    Alarm26 : BOOL ;
    Alarm27 : BOOL ;
    Alarm28 : BOOL ;
    Alarm29 : BOOL ;
    Alarm30 : BOOL ;
    Alarm31 : BOOL ;
    Alarm32 : BOOL ;
    Alarm33 : BOOL ;
    Alarm34 : BOOL ;
    Alarm35 : BOOL ;
    Alarm36 : BOOL ;
    Alarm37 : BOOL ;
    Alarm38 : BOOL ;
    Alarm39 : BOOL ;
    Alarm40 : BOOL ;
    Alarm41 : BOOL ;
    Alarm42 : BOOL ;
    Alarm43 : BOOL ;
    Alarm44 : BOOL ;
    Alarm45 : BOOL ;
    Alarm46 : BOOL ;
    Alarm47 : BOOL ;
    Alarm48 : BOOL ;
    Alarm49 : BOOL ;
    Alarm50 : BOOL ;
    Alarm51 : BOOL ;
    Alarm52 : BOOL ;
    Alarm53 : BOOL ;
    Alarm54 : BOOL ;
    Alarm55 : BOOL ;
    Alarm56 : BOOL ;
    Alarm57 : BOOL ;
    Alarm58 : BOOL ;
    Alarm59 : BOOL ;
    Alarm60 : BOOL ;
    Alarm61 : BOOL ;
    Alarm62 : BOOL ;
    Alarm63 : BOOL ;
    Alarm64 : BOOL ;
   END_STRUCT ;
   StopCycle : STRUCT
    Alarm01 : BOOL ;	//Ribaditrice non bassa
    Alarm02 : BOOL ;	//Ribaditrice non alta
    Alarm03 : BOOL ;	//Incongruenza sensori ribaditrice
    Alarm04 : BOOL ;	//Porte non chiuse
    Alarm05 : BOOL ;	//Chiave non Bloccata Porta SX
    Alarm06 : BOOL ;	//Chiave non Bloccata Porta DX
    Alarm07 : BOOL ;	//asse X bloccato con Ribaditrice non alta
    Alarm08 : BOOL ;	//asse Y bloccato con Ribaditrice non alta
    Alarm09 : BOOL ;
    Alarm10 : BOOL ;
    Alarm11 : BOOL ;	//Macchina in emergenza
    Alarm12 : BOOL ;
    Alarm13 : BOOL ;
    Alarm14 : BOOL ;
    Alarm15 : BOOL ;
    Alarm16 : BOOL ;
    Alarm17 : BOOL ;
    Alarm18 : BOOL ;
    Alarm19 : BOOL ;
    Alarm20 : BOOL ;
    Alarm21 : BOOL ;
    Alarm22 : BOOL ;
    Alarm23 : BOOL ;
    Alarm24 : BOOL ;
    Alarm25 : BOOL ;
    Alarm26 : BOOL ;
    Alarm27 : BOOL ;
    Alarm28 : BOOL ;
    Alarm29 : BOOL ;
    Alarm30 : BOOL ;
    Alarm31 : BOOL ;
    Alarm32 : BOOL ;
    Alarm33 : BOOL ;
    Alarm34 : BOOL ;
    Alarm35 : BOOL ;
    Alarm36 : BOOL ;
    Alarm37 : BOOL ;
    Alarm38 : BOOL ;
    Alarm39 : BOOL ;
    Alarm40 : BOOL ;
    Alarm41 : BOOL ;
    Alarm42 : BOOL ;
    Alarm43 : BOOL ;
    Alarm44 : BOOL ;
    Alarm45 : BOOL ;
    Alarm46 : BOOL ;
    Alarm47 : BOOL ;
    Alarm48 : BOOL ;
    Alarm49 : BOOL ;
    Alarm50 : BOOL ;
    Alarm51 : BOOL ;
    Alarm52 : BOOL ;
    Alarm53 : BOOL ;
    Alarm54 : BOOL ;
    Alarm55 : BOOL ;
    Alarm56 : BOOL ;
    Alarm57 : BOOL ;
    Alarm58 : BOOL ;
    Alarm59 : BOOL ;
    Alarm60 : BOOL ;
    Alarm61 : BOOL ;
    Alarm62 : BOOL ;
    Alarm63 : BOOL ;
    Alarm64 : BOOL ;
   END_STRUCT ;
   RestartCycle : STRUCT
    Alarm01 : BOOL ;
    Alarm02 : BOOL ;
    Alarm03 : BOOL ;
    Alarm04 : BOOL ;
    Alarm05 : BOOL ;
    Alarm06 : BOOL ;
    Alarm07 : BOOL ;
    Alarm08 : BOOL ;
    Alarm09 : BOOL ;
    Alarm10 : BOOL ;
    Alarm11 : BOOL ;
    Alarm12 : BOOL ;
    Alarm13 : BOOL ;
    Alarm14 : BOOL ;
    Alarm15 : BOOL ;
    Alarm16 : BOOL ;
    Alarm17 : BOOL ;
    Alarm18 : BOOL ;
    Alarm19 : BOOL ;
    Alarm20 : BOOL ;
    Alarm21 : BOOL ;
    Alarm22 : BOOL ;
    Alarm23 : BOOL ;
    Alarm24 : BOOL ;
    Alarm25 : BOOL ;
    Alarm26 : BOOL ;
    Alarm27 : BOOL ;
    Alarm28 : BOOL ;
    Alarm29 : BOOL ;
    Alarm30 : BOOL ;
    Alarm31 : BOOL ;
    Alarm32 : BOOL ;
    Alarm33 : BOOL ;
    Alarm34 : BOOL ;
    Alarm35 : BOOL ;
    Alarm36 : BOOL ;
    Alarm37 : BOOL ;
    Alarm38 : BOOL ;
    Alarm39 : BOOL ;
    Alarm40 : BOOL ;
    Alarm41 : BOOL ;
    Alarm42 : BOOL ;
    Alarm43 : BOOL ;
    Alarm44 : BOOL ;
    Alarm45 : BOOL ;
    Alarm46 : BOOL ;
    Alarm47 : BOOL ;
    Alarm48 : BOOL ;
    Alarm49 : BOOL ;
    Alarm50 : BOOL ;
    Alarm51 : BOOL ;
    Alarm52 : BOOL ;
    Alarm53 : BOOL ;
    Alarm54 : BOOL ;
    Alarm55 : BOOL ;
    Alarm56 : BOOL ;
    Alarm57 : BOOL ;
    Alarm58 : BOOL ;
    Alarm59 : BOOL ;
    Alarm60 : BOOL ;
    Alarm61 : BOOL ;
    Alarm62 : BOOL ;
    Alarm63 : BOOL ;
    Alarm64 : BOOL ;
   END_STRUCT ;
   Warning : STRUCT
    Alarm01 : BOOL ;	//Q_Ribaditrice
    Alarm02 : BOOL ;	//Q_Automatici_230_V
    Alarm03 : BOOL ;	//Anomalia_Condizionatore
    Alarm04 : BOOL ;	//Ribaditrice bloccata con motore ribaditrice ferma
    Alarm05 : BOOL ;	//Marcia ribaditrice solo con cassetti OP10 e OP40 indexati
    Alarm06 : BOOL ;	//Dicesa dibaditrice solo con cassetti OP10 e OP40 indexati
    Alarm07 : BOOL ;	//Marcia assi solo con cassetti OP10 e OP40 indexati
    Alarm08 : BOOL ;
    Alarm09 : BOOL ;
    Alarm10 : BOOL ;
    Alarm11 : BOOL ;
    Alarm12 : BOOL ;
    Alarm13 : BOOL ;
    Alarm14 : BOOL ;
    Alarm15 : BOOL ;
    Alarm16 : BOOL ;
    Alarm17 : BOOL ;
    Alarm18 : BOOL ;
    Alarm19 : BOOL ;
    Alarm20 : BOOL ;
    Alarm21 : BOOL ;
    Alarm22 : BOOL ;
    Alarm23 : BOOL ;
    Alarm24 : BOOL ;
    Alarm25 : BOOL ;
    Alarm26 : BOOL ;
    Alarm27 : BOOL ;
    Alarm28 : BOOL ;
    Alarm29 : BOOL ;
    Alarm30 : BOOL ;
    Alarm31 : BOOL ;
    Alarm32 : BOOL ;
    Alarm33 : BOOL ;
    Alarm34 : BOOL ;
    Alarm35 : BOOL ;
    Alarm36 : BOOL ;
    Alarm37 : BOOL ;
    Alarm38 : BOOL ;
    Alarm39 : BOOL ;
    Alarm40 : BOOL ;
    Alarm41 : BOOL ;
    Alarm42 : BOOL ;
    Alarm43 : BOOL ;
    Alarm44 : BOOL ;
    Alarm45 : BOOL ;
    Alarm46 : BOOL ;
    Alarm47 : BOOL ;
    Alarm48 : BOOL ;
    Alarm49 : BOOL ;
    Alarm50 : BOOL ;
    Alarm51 : BOOL ;
    Alarm52 : BOOL ;
    Alarm53 : BOOL ;
    Alarm54 : BOOL ;
    Alarm55 : BOOL ;
    Alarm56 : BOOL ;
    Alarm57 : BOOL ;
    Alarm58 : BOOL ;
    Alarm59 : BOOL ;
    Alarm60 : BOOL ;
    Alarm61 : BOOL ;
    Alarm62 : BOOL ;
    Alarm63 : BOOL ;
    Alarm64 : BOOL ;
   END_STRUCT ;
  END_STRUCT ;	
BEGIN
END_DATA_BLOCK

DATA_BLOCK DB 55
VERSION : 0.1
  STRUCT
   Command : STRUCT 	//
    Reset_allarmi : BOOL ;
    TestLampade : BOOL ;	//da programmare sul pannello operatore
    Abbassa_ribaditrice : BOOL ;
    Alza_ribaditrice : BOOL ;
    Marcia_ribaditrice : BOOL ;	//manca ingresso
    Marcia_manuale_ribaditr : BOOL ;
    Posiziona_Assi : BOOL ;
    ris_0_7 : BOOL ;
    AsseX_Enable : BOOL ;
    AsseX_StartPosizionam : BOOL ;
    AsseX_ris_2 : BOOL ;
    AsseX_ris_3 : BOOL ;
    AsseX_ris_4 : BOOL ;
    AsseX_ris_5 : BOOL ;
    AsseX_ris_6 : BOOL ;
    AsseX_ris_7 : BOOL ;
    AsseY_Enable : BOOL ;
    AsseY_StartPosizionam : BOOL ;
    AsseY_ris_2 : BOOL ;
    AsseY_ris_3 : BOOL ;
    AsseY_ris_4 : BOOL ;
    AsseY_ris_5 : BOOL ;
    AsseY_ris_6 : BOOL ;
    AsseY_ris_7 : BOOL ;
    PrenotaRib_OP10 : BOOL ;
    PrenotaRib_OP40 : BOOL ;
    ris_w4 : WORD ;
    ris_w6 : DWORD ;
   END_STRUCT ;
   State : STRUCT 	//da ind. 10
    PLC_OK : BOOL ;
    Porte_chiuse : BOOL ;
    Ribadit_Motore_in_marcia : BOOL ;
    Ribaditrice_bassa : BOOL ;
    Ribaditrice_alta : BOOL ;
    Porte_chiuse_e_bloccate : BOOL ;
    Cassetto_OP10_indexato : BOOL ;
    Cassetto_OP40_indexato : BOOL ;
    AsseX_referenziato : BOOL ;
    AsseX_posizioneRaggiunta : BOOL ;
    AsseX_inMovimento : BOOL ;
    Ris_1_3 : BOOL ;
    AsseX_ExtracorsaOK : BOOL ;
    AsseX_FC_indietro : BOOL ;
    AsseX_FC_avanti : BOOL ;
    AsseX_Pronto : BOOL ;
    AsseY_referenziato : BOOL ;
    AsseY_posizioneRaggiunta : BOOL ;
    AsseY_inMovimento : BOOL ;
    Ris_2_3 : BOOL ;
    AsseY_ExtracorsaOK : BOOL ;
    AsseY_FC_indietro : BOOL ;
    AsseY_FC_avanti : BOOL ;
    AsseY_pronto : BOOL ;
    Ribad_prenotata_da_OP10 : BOOL ;
    Ribad_prenotata_da_OP40 : BOOL ;
    FP_IngressoInPag_TeachIn : BOOL ;
    FP_NumPuntoCambiato : BOOL ;
    FP_RichiestaLeggiPunto : BOOL ;
    FP_RichiestaSalvaPunto : BOOL ;
    FP_RichiestaTeachInPunto : BOOL ;
    ris_w4 : WORD ;
    ris_w6 : DWORD ;
   END_STRUCT ;
   Data : STRUCT 	//da ind. 20
    ris_X_0 : INT ;
    AsseX_Accelerazione : INT ;
    AsseX_Decellerazione : INT ;
    AsseX_Velocita : DINT ;
    AsseX_PosizioneComandata : DINT ;
    AsseX_PosizioneAttuale : DINT ;
    AsseX_CodiceErrore : BYTE ;
    AsseX_ris20 : WORD ;
    AsseX_ris22 : DWORD ;
    AsseX_ris26 : DWORD ;
    ris_Y_30 : INT ;
    AsseY_Accelerazione : INT ;
    AsseY_Decellerazione : INT ;
    AsseY_Velocita : DINT ;
    AsseY_PosizioneComandata : DINT ;
    AsseY_PosizioneAttuale : DINT ;
    AsseY_CodiceErrore : BYTE ;
    AsseY_ris50 : WORD ;
    AsseY_ris52 : DWORD ;
    AsseY_ris56 : DWORD ;
    PuntoInTeachIn : INT ;
    ris_82 : INT ;
    ris_84 : INT ;
    ris_86 : DINT ;
    ris_90 : ARRAY  [0 .. 40 ] OF INT ;
   END_STRUCT ;
  END_STRUCT ;	
BEGIN
   Command.AsseX_Enable := TRUE;
   Command.AsseY_Enable := TRUE;
   State.PLC_OK := TRUE;
   State.Porte_chiuse := TRUE;
   State.Ribaditrice_alta := TRUE;
   State.Porte_chiuse_e_bloccate := TRUE;
   State.Cassetto_OP10_indexato := TRUE;
   State.Cassetto_OP40_indexato := TRUE;
   State.AsseX_referenziato := TRUE;
   State.AsseX_ExtracorsaOK := TRUE;
   State.AsseX_Pronto := TRUE;
   State.AsseY_referenziato := TRUE;
   State.AsseY_ExtracorsaOK := TRUE;
   State.AsseY_pronto := TRUE;
   Data.AsseX_Accelerazione := 100;
   Data.AsseX_Decellerazione := 100;
   Data.AsseX_Velocita := L#15000;
   Data.AsseX_PosizioneAttuale := L#347483;
   Data.AsseY_Accelerazione := 100;
   Data.AsseY_Decellerazione := 100;
   Data.AsseY_Velocita := L#15000;
   Data.AsseY_PosizioneAttuale := L#23007;
   Data.PuntoInTeachIn := 1;
END_DATA_BLOCK

DATA_BLOCK DB 60
VERSION : 0.1
  STRUCT
   Coord_Ribaditrice : UDT 200;
  END_STRUCT ;	
BEGIN
// 22 bytes; values not shown
END_DATA_BLOCK

DATA_BLOCK DB 70
VERSION : 0.1
  STRUCT
   OP_System_Data : STRUCT
    PageDisplayed : INT ;
    Year_Byte0 : BYTE ;
    Year_Byte1 : BYTE ;
    Month_byte0 : BYTE ;
    Month_byte1 : BYTE ;
    Day_byte0 : BYTE ;
    Day_byte1 : BYTE ;
    HH : BYTE ;
    MM : BYTE ;
    NewPage : INT ;
   END_STRUCT ;
   Commands : STRUCT 	//da indirizzo 12
    Man_Alza_Abb_Ribaditrice : BOOL ;
    Man_Marcia_Ribaditrice : BOOL ;
    Man_Jog_AsseX : BOOL ;
    Man_Jog_AsseY : BOOL ;
    Man_10_IndexCassetto : BOOL ;
    Man_10_BloccoPezzo : BOOL ;
    Man_20_IndexCassetto : BOOL ;
    Man_20_GruppoPiantaggio : BOOL ;
    Man_20_Piantaggio : BOOL ;
    Man_40_IndexCassetto : BOOL ;
    Man_40_BloccoPezzo : BOOL ;
    Man_disp_2_3 : BOOL ;
    Man_disp_2_4 : BOOL ;
    Man_disp_2_5 : BOOL ;
    Man_disp_2_6 : BOOL ;
    Man_disp_2_7 : BOOL ;
    Man_VaiAlPunto : WORD ;
    Reset_Allarmi : BOOL ;
    Cmd_VaiAlPunto : BOOL ;
    Cmd_TeachInPunto : BOOL ;
    Cmd_SalvaPunto : BOOL ;
    Cmd_LeggiPunto : BOOL ;
    Ris_16_5 : BOOL ;
    ris_w18 : DINT ;
    ris_w22 : DINT ;
   END_STRUCT ;
   States : STRUCT 	//da indirizzo 26
    RibaditriceAlta : BOOL ;
    RibaditriceBassa : BOOL ;
    RibaditriceFerma : BOOL ;
    RibaditriceInMarcia : BOOL ;
    OP10IndexCassSbloccato : BOOL ;
    OP10IndexCassBloccato : BOOL ;
    OP10PezzoSbloccato : BOOL ;
    OP10PezzoBloccato : BOOL ;
    AsseXIndietro : BOOL ;
    AsseXAvanti : BOOL ;
    AsseYIndietro : BOOL ;
    AsseYAvanti : BOOL ;
    OP20IndexCassSbloccato : BOOL ;
    OP20IndexCassBloccato : BOOL ;
    OP20GrPiantaggioAlto : BOOL ;
    OP20GrPiantaggioBasso : BOOL ;
    OP20PiantaggioAlto : BOOL ;
    OP20PiantaggioBasso : BOOL ;
    OP40IndexCassSbloccato : BOOL ;
    OP40IndexCassBloccato : BOOL ;
    OP40PezzoSbloccato : BOOL ;
    OP40PezzoBloccato : BOOL ;
    ris_w30 : INT ;
    ris_w32 : DINT ;
   END_STRUCT ;
   Data : STRUCT 	//da indirizzo 36
    AsseX_PosizioneAttuale : DINT ;	//Valori assoluti assi
    AsseY_PosizioneAttuale : DINT ;	//Valori assoluti assi
    PosizionePunzone : REAL ;
    Cmd_Override_man : INT ;
    Cmd_Override_auto : INT ;
    AsseX_PosAttualeOP10 : DINT ;
    AsseY_PosAttualeOP10 : DINT ;
    AsseX_PosAttualeOP40 : DINT ;
    AsseY_PosAttualeOP40 : DINT ;
    Cmd_PuntoSelezionato : INT ;
    Min_PerSelezionePunto : INT ;
    Max_PerSelezionePunto : INT ;
    X_PosPuntoSelezionato : DINT ;
    Y_PosPuntoSelezionato : DINT ;
    TempoRibad_PuntoSelez : DINT ;
    ris_array : ARRAY  [0 .. 15 ] OF REAL ;
   END_STRUCT ;
   cycles : STRUCT 	//indirizzo 150
    OP10_cycle_general : BOOL ;
    OP10_cycle_restore : BOOL ;
    OP20_cycle_general : BOOL ;
    OP20_cycle_restore : BOOL ;
    OP40_cycle_general : BOOL ;
    OP40_cycle_restore : BOOL ;
    OP10_message : INT ;
    OP10_spacer : INT ;
    OP40_message : INT ;
    OP40_spacer : INT ;
    OP20_message : INT ;
    Line_State : INT ;
    ris_w8 : INT ;
    ris_array : ARRAY  [0 .. 16 ] OF INT ;
   END_STRUCT ;
  END_STRUCT ;	
BEGIN
   OP_System_Data.PageDisplayed := 120;
   OP_System_Data.Year_Byte1 := B#16#10;
   OP_System_Data.Month_byte1 := B#16#4;
   OP_System_Data.Day_byte1 := B#16#6;
   OP_System_Data.HH := B#16#21;
   OP_System_Data.MM := B#16#39;
   OP_System_Data.NewPage := 120;
   Commands.Man_Marcia_Ribaditrice := TRUE;
   States.RibaditriceAlta := TRUE;
   States.RibaditriceFerma := TRUE;
   States.OP10IndexCassBloccato := TRUE;
   States.OP10PezzoBloccato := TRUE;
   States.OP20IndexCassSbloccato := TRUE;
   States.OP20GrPiantaggioAlto := TRUE;
   States.OP20PiantaggioAlto := TRUE;
   States.OP40IndexCassBloccato := TRUE;
   States.OP40PezzoSbloccato := TRUE;
   Data.AsseX_PosizioneAttuale := L#347483;
   Data.AsseY_PosizioneAttuale := L#23007;
   Data.PosizionePunzone := -3.808000e+00;
   Data.Cmd_Override_man := 100;
   Data.Cmd_Override_auto := 40;
   Data.AsseX_PosAttualeOP10 := L#275982;
   Data.AsseY_PosAttualeOP10 := L#-24109;
   Data.AsseX_PosAttualeOP40 := L#-24040;
   Data.AsseY_PosAttualeOP40 := L#-24040;
   Data.Cmd_PuntoSelezionato := 1;
   Data.Min_PerSelezionePunto := 1;
   Data.Max_PerSelezionePunto := 1;
   Data.X_PosPuntoSelezionato := L#-24040;
   Data.Y_PosPuntoSelezionato := L#-24040;
   Data.TempoRibad_PuntoSelez := L#3000;
   cycles.OP10_cycle_general := TRUE;
   cycles.OP20_cycle_general := TRUE;
   cycles.OP40_cycle_general := TRUE;
   cycles.OP10_message := 2;
   cycles.OP40_message := 4;
   cycles.OP20_message := 2;
   cycles.Line_State := 4;
END_DATA_BLOCK

DATA_BLOCK DB 100
VERSION : 0.1
UDT 250
BEGIN
END_DATA_BLOCK

DATA_BLOCK DB 101
VERSION : 0.1
  STRUCT
   P_Consenso_operatore : BOOL ;	//(start ciclo)
   Cassetto_fuori : BOOL ;
   Cassetto_dentro : BOOL ;
   Index_cassetto_Giu : BOOL ;
   Index_cassetto_Su : BOOL ;
   Sblocco_pezzo_Giu : BOOL ;
   Sblocco_pezzo_Su : BOOL ;
   PulStopCiclo : BOOL ;
  END_STRUCT ;	
BEGIN
   Cassetto_fuori := TRUE;
   Index_cassetto_Su := TRUE;
   Sblocco_pezzo_Su := TRUE;
END_DATA_BLOCK

DATA_BLOCK DB 102
VERSION : 0.1
  STRUCT
   Fine_ciclo_OK : BOOL ;	//
   Fine_ciclo_NON_OK : BOOL ;
   EV_abb_index_cassetto : BOOL ;
   EV_alza_index_cassetto : BOOL ;
   EV_sblocco_pezzo : BOOL ;
   EV_blocco_pezzo : BOOL ;	//??? esiste?
  END_STRUCT ;	
BEGIN
   EV_alza_index_cassetto := TRUE;
   EV_sblocco_pezzo := TRUE;
END_DATA_BLOCK

DATA_BLOCK DB 103
VERSION : 0.1
  STRUCT
   dummy : INT ;
  END_STRUCT ;	
BEGIN
END_DATA_BLOCK

DATA_BLOCK DB 104
VERSION : 0.1
  STRUCT
   Emegency : STRUCT
    Alarm01 : BOOL ;	//OP10 ToolType error
    Alarm02 : BOOL ;	//OP10 ToolCode error
    Alarm03 : BOOL ;
    Alarm04 : BOOL ;
    Alarm05 : BOOL ;
    Alarm06 : BOOL ;
    Alarm07 : BOOL ;
    Alarm08 : BOOL ;
    Alarm09 : BOOL ;	//
    Alarm10 : BOOL ;	//
    Alarm11 : BOOL ;	//
    Alarm12 : BOOL ;	//
    Alarm13 : BOOL ;	//
    Alarm14 : BOOL ;	//
    Alarm15 : BOOL ;
    Alarm16 : BOOL ;
    Alarm17 : BOOL ;
    Alarm18 : BOOL ;
    Alarm19 : BOOL ;
    Alarm20 : BOOL ;
    Alarm21 : BOOL ;
    Alarm22 : BOOL ;
    Alarm23 : BOOL ;
    Alarm24 : BOOL ;
    Alarm25 : BOOL ;
    Alarm26 : BOOL ;
    Alarm27 : BOOL ;
    Alarm28 : BOOL ;
    Alarm29 : BOOL ;
    Alarm30 : BOOL ;
    Alarm31 : BOOL ;
    Alarm32 : BOOL ;
    Alarm33 : BOOL ;
    Alarm34 : BOOL ;
    Alarm35 : BOOL ;
    Alarm36 : BOOL ;
    Alarm37 : BOOL ;
    Alarm38 : BOOL ;
    Alarm39 : BOOL ;
    Alarm40 : BOOL ;
    Alarm41 : BOOL ;
    Alarm42 : BOOL ;
    Alarm43 : BOOL ;
    Alarm44 : BOOL ;
    Alarm45 : BOOL ;
    Alarm46 : BOOL ;
    Alarm47 : BOOL ;
    Alarm48 : BOOL ;
    Alarm49 : BOOL ;
    Alarm50 : BOOL ;
    Alarm51 : BOOL ;
    Alarm52 : BOOL ;
    Alarm53 : BOOL ;
    Alarm54 : BOOL ;
    Alarm55 : BOOL ;
    Alarm56 : BOOL ;
    Alarm57 : BOOL ;
    Alarm58 : BOOL ;
    Alarm59 : BOOL ;
    Alarm60 : BOOL ;
    Alarm61 : BOOL ;
    Alarm62 : BOOL ;
    Alarm63 : BOOL ;
    Alarm64 : BOOL ;
   END_STRUCT ;
   StopCycle : STRUCT
    Alarm01 : BOOL ;	//Errore rilevamento anello di adattamento 1
    Alarm02 : BOOL ;	//Errore rilevamento anello di adattamento 2
    Alarm03 : BOOL ;	//Index cassetto non alto
    Alarm04 : BOOL ;	//Index cassetto non basso
    Alarm05 : BOOL ;	//Incongruenza sensori index cassetto
    Alarm06 : BOOL ;	//Cilindro sblocco pezzo non avanti
    Alarm07 : BOOL ;	//Cilindro sblocco pezzo non indietro
    Alarm08 : BOOL ;	//Incongruenza sensori cilindro sblocco pezzo
    Alarm09 : BOOL ;	//OP10 ToolType error
    Alarm10 : BOOL ;	//OP10 ToolCode error
    Alarm11 : BOOL ;
    Alarm12 : BOOL ;
    Alarm13 : BOOL ;
    Alarm14 : BOOL ;
    Alarm15 : BOOL ;
    Alarm16 : BOOL ;
    Alarm17 : BOOL ;
    Alarm18 : BOOL ;
    Alarm19 : BOOL ;
    Alarm20 : BOOL ;
    Alarm21 : BOOL ;
    Alarm22 : BOOL ;
    Alarm23 : BOOL ;
    Alarm24 : BOOL ;
    Alarm25 : BOOL ;
    Alarm26 : BOOL ;
    Alarm27 : BOOL ;
    Alarm28 : BOOL ;
    Alarm29 : BOOL ;
    Alarm30 : BOOL ;
    Alarm31 : BOOL ;
    Alarm32 : BOOL ;
    Alarm33 : BOOL ;
    Alarm34 : BOOL ;
    Alarm35 : BOOL ;
    Alarm36 : BOOL ;
    Alarm37 : BOOL ;
    Alarm38 : BOOL ;
    Alarm39 : BOOL ;
    Alarm40 : BOOL ;
    Alarm41 : BOOL ;
    Alarm42 : BOOL ;
    Alarm43 : BOOL ;
    Alarm44 : BOOL ;
    Alarm45 : BOOL ;
    Alarm46 : BOOL ;
    Alarm47 : BOOL ;
    Alarm48 : BOOL ;
    Alarm49 : BOOL ;
    Alarm50 : BOOL ;
    Alarm51 : BOOL ;
    Alarm52 : BOOL ;
    Alarm53 : BOOL ;
    Alarm54 : BOOL ;
    Alarm55 : BOOL ;
    Alarm56 : BOOL ;
    Alarm57 : BOOL ;
    Alarm58 : BOOL ;
    Alarm59 : BOOL ;
    Alarm60 : BOOL ;
    Alarm61 : BOOL ;
    Alarm62 : BOOL ;
    Alarm63 : BOOL ;
    Alarm64 : BOOL ;
   END_STRUCT ;
   RestartCycle : STRUCT
    Alarm01 : BOOL ;
    Alarm02 : BOOL ;
    Alarm03 : BOOL ;
    Alarm04 : BOOL ;
    Alarm05 : BOOL ;
    Alarm06 : BOOL ;
    Alarm07 : BOOL ;
    Alarm08 : BOOL ;
    Alarm09 : BOOL ;
    Alarm10 : BOOL ;
    Alarm11 : BOOL ;
    Alarm12 : BOOL ;
    Alarm13 : BOOL ;
    Alarm14 : BOOL ;
    Alarm15 : BOOL ;
    Alarm16 : BOOL ;
    Alarm17 : BOOL ;
    Alarm18 : BOOL ;
    Alarm19 : BOOL ;
    Alarm20 : BOOL ;
    Alarm21 : BOOL ;
    Alarm22 : BOOL ;
    Alarm23 : BOOL ;
    Alarm24 : BOOL ;
    Alarm25 : BOOL ;
    Alarm26 : BOOL ;
    Alarm27 : BOOL ;
    Alarm28 : BOOL ;
    Alarm29 : BOOL ;
    Alarm30 : BOOL ;
    Alarm31 : BOOL ;
    Alarm32 : BOOL ;
    Alarm33 : BOOL ;
    Alarm34 : BOOL ;
    Alarm35 : BOOL ;
    Alarm36 : BOOL ;
    Alarm37 : BOOL ;
    Alarm38 : BOOL ;
    Alarm39 : BOOL ;
    Alarm40 : BOOL ;
    Alarm41 : BOOL ;
    Alarm42 : BOOL ;
    Alarm43 : BOOL ;
    Alarm44 : BOOL ;
    Alarm45 : BOOL ;
    Alarm46 : BOOL ;
    Alarm47 : BOOL ;
    Alarm48 : BOOL ;
    Alarm49 : BOOL ;
    Alarm50 : BOOL ;
    Alarm51 : BOOL ;
    Alarm52 : BOOL ;
    Alarm53 : BOOL ;
    Alarm54 : BOOL ;
    Alarm55 : BOOL ;
    Alarm56 : BOOL ;
    Alarm57 : BOOL ;
    Alarm58 : BOOL ;
    Alarm59 : BOOL ;
    Alarm60 : BOOL ;
    Alarm61 : BOOL ;
    Alarm62 : BOOL ;
    Alarm63 : BOOL ;
    Alarm64 : BOOL ;
   END_STRUCT ;
   Warning : STRUCT
    Alarm01 : BOOL ;	//Blocco movimento index cassetto se cassetto non dentro o non fuori
    Alarm02 : BOOL ;	//Blocco sblocco pezzo se cassetto non fuori
    Alarm03 : BOOL ;	//Sblocco index solo con ribaditrice alta
    Alarm04 : BOOL ;	//Sblocco index solo con assi fermi
    Alarm05 : BOOL ;	//Sblocco index solo pezzo bloccato
    Alarm06 : BOOL ;
    Alarm07 : BOOL ;
    Alarm08 : BOOL ;
    Alarm09 : BOOL ;
    Alarm10 : BOOL ;
    Alarm11 : BOOL ;
    Alarm12 : BOOL ;
    Alarm13 : BOOL ;
    Alarm14 : BOOL ;
    Alarm15 : BOOL ;
    Alarm16 : BOOL ;
    Alarm17 : BOOL ;
    Alarm18 : BOOL ;
    Alarm19 : BOOL ;
    Alarm20 : BOOL ;
    Alarm21 : BOOL ;
    Alarm22 : BOOL ;
    Alarm23 : BOOL ;
    Alarm24 : BOOL ;
    Alarm25 : BOOL ;
    Alarm26 : BOOL ;
    Alarm27 : BOOL ;
    Alarm28 : BOOL ;
    Alarm29 : BOOL ;
    Alarm30 : BOOL ;
    Alarm31 : BOOL ;
    Alarm32 : BOOL ;
    Alarm33 : BOOL ;
    Alarm34 : BOOL ;
    Alarm35 : BOOL ;
    Alarm36 : BOOL ;
    Alarm37 : BOOL ;
    Alarm38 : BOOL ;
    Alarm39 : BOOL ;
    Alarm40 : BOOL ;
    Alarm41 : BOOL ;
    Alarm42 : BOOL ;
    Alarm43 : BOOL ;
    Alarm44 : BOOL ;
    Alarm45 : BOOL ;
    Alarm46 : BOOL ;
    Alarm47 : BOOL ;
    Alarm48 : BOOL ;
    Alarm49 : BOOL ;
    Alarm50 : BOOL ;
    Alarm51 : BOOL ;
    Alarm52 : BOOL ;
    Alarm53 : BOOL ;
    Alarm54 : BOOL ;
    Alarm55 : BOOL ;
    Alarm56 : BOOL ;
    Alarm57 : BOOL ;
    Alarm58 : BOOL ;
    Alarm59 : BOOL ;
    Alarm60 : BOOL ;
    Alarm61 : BOOL ;
    Alarm62 : BOOL ;
    Alarm63 : BOOL ;
    Alarm64 : BOOL ;
   END_STRUCT ;
  END_STRUCT ;	
BEGIN
   Warning.Alarm05 := TRUE;
END_DATA_BLOCK

DATA_BLOCK DB 105
VERSION : 0.1
  STRUCT
   Command : STRUCT 	//
    Reset_allarmi : BOOL ;
    TestLampade : BOOL ;
    Abbassa_index_cassetto : BOOL ;
    Alza_index_cassetto : BOOL ;
    Sblocca_pezzo : BOOL ;
    Blocca_pezzo : BOOL ;
    FP_Consenso_operatore : BOOL ;
    Prenota_ribaditrice : BOOL ;
    Vai_in_posizione_assi : BOOL ;
    Marcia_ribaditrice : BOOL ;
    Abbassa_ribaditrice : BOOL ;
    Alza_ribaditrice : BOOL ;
    ris_w2 : DWORD ;
    ris_w6 : DWORD ;
   END_STRUCT ;
   State : STRUCT
    Porte_chiuse : BOOL ;
    Porte_chiuse_e_bloccate : BOOL ;
    Cassetto_dentro : BOOL ;
    Cassetto_fuori : BOOL ;
    Index_cassetto_basso : BOOL ;
    Index_cassetto_alto : BOOL ;
    Pezzo_sbloccato : BOOL ;
    Pezzo_bloccato : BOOL ;
    _Ribaditrice_a_disposiz : BOOL ;
    _Assi_posiz_raggiunta : BOOL ;
    Ribaditura_effettuata : BOOL ;
    Ribaditrice_alta : BOOL ;
    Ribaditrice_bassa : BOOL ;
    Ribaditrice_in_marcia : BOOL ;
    FP_stato_20_generale : BOOL ;
    _Ribad_in_fuori_ingombro : BOOL ;
    FP_Mode_automatic : BOOL ;
    FP_uscita_da_allarme : BOOL ;
    Ribaditura_pezzo_OK : BOOL ;
    Ribaditura_pezzo_KO : BOOL ;
    Assi_fermi : BOOL ;
    ris_w4 : WORD ;
    ris_w6 : DWORD ;
   END_STRUCT ;
   Data : STRUCT
    Num_punto_in_lavorazione : INT ;
    Pos_comandata_asse_X : DINT ;	//Punto in lavorazione
    Pos_comandata_asse_Y : DINT ;	//Punto in lavorazione
    Tempo_ribaditura : DINT ;	//Punto in lavorazione
    ris_w2 : DWORD ;
    ris_w6 : DWORD ;
   END_STRUCT ;
  END_STRUCT ;	
BEGIN
   State.Porte_chiuse := TRUE;
   State.Porte_chiuse_e_bloccate := TRUE;
   State.Cassetto_fuori := TRUE;
   State.Index_cassetto_alto := TRUE;
   State.Pezzo_bloccato := TRUE;
   State.Ribaditrice_alta := TRUE;
   State.Assi_fermi := TRUE;
END_DATA_BLOCK

DATA_BLOCK DB 106
VERSION : 0.1
  STRUCT
   ToolCode_Bit_0 : BOOL ;	//
   ToolCode_Bit_1 : BOOL ;
   ToolCode_Bit_2 : BOOL ;
   ToolCode_Bit_3 : BOOL ;
   ToolCode_Bit_4 : BOOL ;
   Anello_1_Inserito : BOOL ;
   Anello_2_Inserito : BOOL ;
   Presenza_nozzle_ring : BOOL ;
   Spacer_1_presente : BOOL ;
   Spacer_1_invertito : BOOL ;
   Spacer_2_presente : BOOL ;
   Spacer_2_invertito : BOOL ;
   Spacer_3_presente : BOOL ;
   Spacer_3_invertito : BOOL ;
   Ris_1_6 : BOOL ;
   Ris_1_7 : BOOL ;
  END_STRUCT ;	
BEGIN
   ToolCode_Bit_1 := TRUE;
   Anello_1_Inserito := TRUE;
END_DATA_BLOCK

DATA_BLOCK DB 108
VERSION : 0.1
  STRUCT
   DB_VAR : INT ;	//Variabile jolly provvisoria
  END_STRUCT ;	
BEGIN
END_DATA_BLOCK

DATA_BLOCK DB 110
VERSION : 0.1
  STRUCT
   ID_Ricetta : INT ;
   PartNumber : ARRAY  [0 .. 31 ] OF //Part number in lavorazione
   CHAR ;
   ToolType : INT ;	//Tool type
   ToolCode : INT ;	//Codice su attrezzo - ingressi digitali
   Anello1Abilitato : BOOL ;
   Anello2Abilitato : BOOL ;
   Velocita_asse_X : DINT ;
   Velocita_asse_Y : DINT ;
   spare48 : DINT ;
   spare52 : DINT ;
   spare56 : DINT ;
   spare60 : DINT ;
   spare64 : DINT ;
   spare68 : DINT ;
   spare72 : DINT ;
   spare76 : INT ;
   Disable : STRUCT 	//da indirizzo 78
    CkCodicePortapezzo : BOOL ;
    CkPresAnelloAdattamento : BOOL ;
    CkPresenzaNozzleRing : BOOL ;
    CkPresenzaSpacer1 : BOOL ;
    CkPresenzaSpacer2 : BOOL ;
    CkPresenzaSpacer3 : BOOL ;
    CheckSpare1 : BOOL ;
    CheckSpare2 : BOOL ;
    CheckSpare3 : BOOL ;
    CheckSpare4 : BOOL ;
   END_STRUCT ;
   NumeroPosizioni : INT ;
   posizioni : ARRAY  [0 .. 19 ] OF //da indirizzo 82
   STRUCT
    X : DINT ;	//1/100 mm
    Y : DINT ;	//1/100 mm
    TempoRibaditura : DINT ;	//msec
   END_STRUCT ;
   spare : ARRAY  [0 .. 38 ] OF INT ;
  END_STRUCT ;	
BEGIN
   ID_Ricetta := 1;
   PartNumber[0] := 'R';
   PartNumber[1] := 'P';
   PartNumber[2] := 'V';
   PartNumber[3] := 'O';
   PartNumber[4] := ' ';
   PartNumber[5] := 'A';
   PartNumber[6] := 'P';
   PartNumber[7] := 'O';
   PartNumber[8] := '0';
   PartNumber[9] := '1';
   PartNumber[10] := ' ';
   PartNumber[11] := ' ';
   PartNumber[12] := ' ';
   PartNumber[13] := ' ';
   PartNumber[14] := ' ';
   PartNumber[15] := ' ';
   PartNumber[16] := ' ';
   PartNumber[17] := ' ';
   PartNumber[18] := ' ';
   PartNumber[19] := ' ';
   PartNumber[20] := ' ';
   PartNumber[21] := ' ';
   PartNumber[22] := ' ';
   PartNumber[23] := ' ';
   PartNumber[24] := ' ';
   PartNumber[25] := ' ';
   PartNumber[26] := ' ';
   PartNumber[27] := ' ';
   PartNumber[28] := ' ';
   PartNumber[29] := ' ';
   PartNumber[30] := ' ';
   PartNumber[31] := ' ';
   ToolType := 1;
   ToolCode := 2;
   Anello1Abilitato := TRUE;
   Velocita_asse_X := L#100000;
   Velocita_asse_Y := L#100000;
   NumeroPosizioni := 3;
   posizioni[0].X := L#-24040;
   posizioni[0].Y := L#-24040;
   posizioni[0].TempoRibaditura := L#3000;
   posizioni[1].X := L#-15440;
   posizioni[1].Y := L#30290;
   posizioni[1].TempoRibaditura := L#3000;
   posizioni[2].X := L#33580;
   posizioni[2].Y := L#5320;
   posizioni[2].TempoRibaditura := L#3000;
END_DATA_BLOCK

DATA_BLOCK DB 120
VERSION : 0.1
  STRUCT
   General : UDT 200;
   Restore : UDT 200;
  END_STRUCT ;	
BEGIN
// 44 bytes; values not shown
END_DATA_BLOCK

DATA_BLOCK DB 150
VERSION : 0.1
UDT 250
BEGIN
END_DATA_BLOCK

DATA_BLOCK DB 151
VERSION : 0.1
  STRUCT
   Ris_0_0 : BOOL ;
   Ris_0_1 : BOOL ;
   Cassetto_dentro : BOOL ;	//manca ingresso
   Index_cassetto_Giu : BOOL ;	//manca ingresso
   Index_cassetto_Su : BOOL ;	//manca ingresso
   Piantaggio_Giu : BOOL ;
   Piantaggio_Su : BOOL ;
   Gruppo_piantaggio_Giu : BOOL ;
   Gruppo_piantaggio_Su : BOOL ;
   Ris_w2 : WORD ;
   ris_w3 : WORD ;
   _Posizione_Punzone : REAL ;	//mm
  END_STRUCT ;	
BEGIN
   Cassetto_dentro := TRUE;
   Index_cassetto_Giu := TRUE;
   Piantaggio_Su := TRUE;
   Gruppo_piantaggio_Su := TRUE;
   _Posizione_Punzone := -3.808000e+00;
END_DATA_BLOCK

DATA_BLOCK DB 152
VERSION : 0.1
  STRUCT
   Fine_ciclo_OK : BOOL ;	//
   Fine_ciclo_NON_OK : BOOL ;
   EV_abb_index_cassetto : BOOL ;	//Libera index cassetto su zona piantaggio
   EV_alza_index_cassetto : BOOL ;	//Blocca index cassetto su zona piantaggio
   EV_abbassa_piantaggio : BOOL ;
   EV_alza_piantaggio : BOOL ;
   EV_abb_grupp_piantaggio : BOOL ;
   EV_alz_grupp_piantaggio : BOOL ;
  END_STRUCT ;	
BEGIN
   Fine_ciclo_OK := TRUE;
   EV_abb_index_cassetto := TRUE;
   EV_alza_piantaggio := TRUE;
   EV_alz_grupp_piantaggio := TRUE;
END_DATA_BLOCK

DATA_BLOCK DB 153
VERSION : 0.1
  STRUCT
   Offset_Tastatore : REAL ;	//
  END_STRUCT ;	
BEGIN
   Offset_Tastatore := 3.808000e+00;
END_DATA_BLOCK

DATA_BLOCK DB 154
VERSION : 0.1
  STRUCT
   Emegency : STRUCT
    Alarm01 : BOOL ;	//OP20 ToolType error
    Alarm02 : BOOL ;	//OP20 ToolCode error
    Alarm03 : BOOL ;
    Alarm04 : BOOL ;
    Alarm05 : BOOL ;
    Alarm06 : BOOL ;
    Alarm07 : BOOL ;
    Alarm08 : BOOL ;
    Alarm09 : BOOL ;	//
    Alarm10 : BOOL ;	//
    Alarm11 : BOOL ;	//
    Alarm12 : BOOL ;	//
    Alarm13 : BOOL ;	//
    Alarm14 : BOOL ;	//
    Alarm15 : BOOL ;
    Alarm16 : BOOL ;
    Alarm17 : BOOL ;
    Alarm18 : BOOL ;
    Alarm19 : BOOL ;
    Alarm20 : BOOL ;
    Alarm21 : BOOL ;
    Alarm22 : BOOL ;
    Alarm23 : BOOL ;
    Alarm24 : BOOL ;
    Alarm25 : BOOL ;
    Alarm26 : BOOL ;
    Alarm27 : BOOL ;
    Alarm28 : BOOL ;
    Alarm29 : BOOL ;
    Alarm30 : BOOL ;
    Alarm31 : BOOL ;
    Alarm32 : BOOL ;
    Alarm33 : BOOL ;
    Alarm34 : BOOL ;
    Alarm35 : BOOL ;
    Alarm36 : BOOL ;
    Alarm37 : BOOL ;
    Alarm38 : BOOL ;
    Alarm39 : BOOL ;
    Alarm40 : BOOL ;
    Alarm41 : BOOL ;
    Alarm42 : BOOL ;
    Alarm43 : BOOL ;
    Alarm44 : BOOL ;
    Alarm45 : BOOL ;
    Alarm46 : BOOL ;
    Alarm47 : BOOL ;
    Alarm48 : BOOL ;
    Alarm49 : BOOL ;
    Alarm50 : BOOL ;
    Alarm51 : BOOL ;
    Alarm52 : BOOL ;
    Alarm53 : BOOL ;
    Alarm54 : BOOL ;
    Alarm55 : BOOL ;
    Alarm56 : BOOL ;
    Alarm57 : BOOL ;
    Alarm58 : BOOL ;
    Alarm59 : BOOL ;
    Alarm60 : BOOL ;
    Alarm61 : BOOL ;
    Alarm62 : BOOL ;
    Alarm63 : BOOL ;
    Alarm64 : BOOL ;
   END_STRUCT ;
   StopCycle : STRUCT
    Alarm01 : BOOL ;	//Gruppo di piantaggio non basso
    Alarm02 : BOOL ;	//Gruppo di piantaggio non alto
    Alarm03 : BOOL ;	//Incongruenza sensori gruppo di piantaggio
    Alarm04 : BOOL ;	//piantaggio non basso
    Alarm05 : BOOL ;	//piantaggio non alto
    Alarm06 : BOOL ;	//Incongruenza sensori piantaggio
    Alarm07 : BOOL ;	//OP20 ToolType error
    Alarm08 : BOOL ;	//OP20 ToolCode error
    Alarm09 : BOOL ;
    Alarm10 : BOOL ;
    Alarm11 : BOOL ;
    Alarm12 : BOOL ;
    Alarm13 : BOOL ;
    Alarm14 : BOOL ;
    Alarm15 : BOOL ;
    Alarm16 : BOOL ;
    Alarm17 : BOOL ;
    Alarm18 : BOOL ;
    Alarm19 : BOOL ;
    Alarm20 : BOOL ;
    Alarm21 : BOOL ;
    Alarm22 : BOOL ;
    Alarm23 : BOOL ;
    Alarm24 : BOOL ;
    Alarm25 : BOOL ;
    Alarm26 : BOOL ;
    Alarm27 : BOOL ;
    Alarm28 : BOOL ;
    Alarm29 : BOOL ;
    Alarm30 : BOOL ;
    Alarm31 : BOOL ;
    Alarm32 : BOOL ;
    Alarm33 : BOOL ;
    Alarm34 : BOOL ;
    Alarm35 : BOOL ;
    Alarm36 : BOOL ;
    Alarm37 : BOOL ;
    Alarm38 : BOOL ;
    Alarm39 : BOOL ;
    Alarm40 : BOOL ;
    Alarm41 : BOOL ;
    Alarm42 : BOOL ;
    Alarm43 : BOOL ;
    Alarm44 : BOOL ;
    Alarm45 : BOOL ;
    Alarm46 : BOOL ;
    Alarm47 : BOOL ;
    Alarm48 : BOOL ;
    Alarm49 : BOOL ;
    Alarm50 : BOOL ;
    Alarm51 : BOOL ;
    Alarm52 : BOOL ;
    Alarm53 : BOOL ;
    Alarm54 : BOOL ;
    Alarm55 : BOOL ;
    Alarm56 : BOOL ;
    Alarm57 : BOOL ;
    Alarm58 : BOOL ;
    Alarm59 : BOOL ;
    Alarm60 : BOOL ;
    Alarm61 : BOOL ;
    Alarm62 : BOOL ;
    Alarm63 : BOOL ;
    Alarm64 : BOOL ;
   END_STRUCT ;
   RestartCycle : STRUCT
    Alarm01 : BOOL ;
    Alarm02 : BOOL ;
    Alarm03 : BOOL ;
    Alarm04 : BOOL ;
    Alarm05 : BOOL ;
    Alarm06 : BOOL ;
    Alarm07 : BOOL ;
    Alarm08 : BOOL ;
    Alarm09 : BOOL ;
    Alarm10 : BOOL ;
    Alarm11 : BOOL ;
    Alarm12 : BOOL ;
    Alarm13 : BOOL ;
    Alarm14 : BOOL ;
    Alarm15 : BOOL ;
    Alarm16 : BOOL ;
    Alarm17 : BOOL ;
    Alarm18 : BOOL ;
    Alarm19 : BOOL ;
    Alarm20 : BOOL ;
    Alarm21 : BOOL ;
    Alarm22 : BOOL ;
    Alarm23 : BOOL ;
    Alarm24 : BOOL ;
    Alarm25 : BOOL ;
    Alarm26 : BOOL ;
    Alarm27 : BOOL ;
    Alarm28 : BOOL ;
    Alarm29 : BOOL ;
    Alarm30 : BOOL ;
    Alarm31 : BOOL ;
    Alarm32 : BOOL ;
    Alarm33 : BOOL ;
    Alarm34 : BOOL ;
    Alarm35 : BOOL ;
    Alarm36 : BOOL ;
    Alarm37 : BOOL ;
    Alarm38 : BOOL ;
    Alarm39 : BOOL ;
    Alarm40 : BOOL ;
    Alarm41 : BOOL ;
    Alarm42 : BOOL ;
    Alarm43 : BOOL ;
    Alarm44 : BOOL ;
    Alarm45 : BOOL ;
    Alarm46 : BOOL ;
    Alarm47 : BOOL ;
    Alarm48 : BOOL ;
    Alarm49 : BOOL ;
    Alarm50 : BOOL ;
    Alarm51 : BOOL ;
    Alarm52 : BOOL ;
    Alarm53 : BOOL ;
    Alarm54 : BOOL ;
    Alarm55 : BOOL ;
    Alarm56 : BOOL ;
    Alarm57 : BOOL ;
    Alarm58 : BOOL ;
    Alarm59 : BOOL ;
    Alarm60 : BOOL ;
    Alarm61 : BOOL ;
    Alarm62 : BOOL ;
    Alarm63 : BOOL ;
    Alarm64 : BOOL ;
   END_STRUCT ;
   Warning : STRUCT
    Alarm01 : BOOL ;	//Blocco movimento index cassetto se cassetto non dentro
    Alarm02 : BOOL ;	//Index cassetto non alto
    Alarm03 : BOOL ;	//Index cassetto non basso
    Alarm04 : BOOL ;	//Incongruenza sensori index cassetto
    Alarm05 : BOOL ;	//Blocco movimento index cassetto con Pinataggio non alto
    Alarm06 : BOOL ;	//Blocco discesa Piantaggio con cassetto non dentro
    Alarm07 : BOOL ;	//Blocco discesa Piantaggio con cassetto non indexato
    Alarm08 : BOOL ;	//Blocco discesa Piantaggio con gruppo non basso
    Alarm09 : BOOL ;	//Blocco salita Gr Piantaggio se Piantaggio non alto
    Alarm10 : BOOL ;
    Alarm11 : BOOL ;
    Alarm12 : BOOL ;
    Alarm13 : BOOL ;
    Alarm14 : BOOL ;
    Alarm15 : BOOL ;
    Alarm16 : BOOL ;
    Alarm17 : BOOL ;
    Alarm18 : BOOL ;
    Alarm19 : BOOL ;
    Alarm20 : BOOL ;
    Alarm21 : BOOL ;
    Alarm22 : BOOL ;
    Alarm23 : BOOL ;
    Alarm24 : BOOL ;
    Alarm25 : BOOL ;
    Alarm26 : BOOL ;
    Alarm27 : BOOL ;
    Alarm28 : BOOL ;
    Alarm29 : BOOL ;
    Alarm30 : BOOL ;
    Alarm31 : BOOL ;
    Alarm32 : BOOL ;
    Alarm33 : BOOL ;
    Alarm34 : BOOL ;
    Alarm35 : BOOL ;
    Alarm36 : BOOL ;
    Alarm37 : BOOL ;
    Alarm38 : BOOL ;
    Alarm39 : BOOL ;
    Alarm40 : BOOL ;
    Alarm41 : BOOL ;
    Alarm42 : BOOL ;
    Alarm43 : BOOL ;
    Alarm44 : BOOL ;
    Alarm45 : BOOL ;
    Alarm46 : BOOL ;
    Alarm47 : BOOL ;
    Alarm48 : BOOL ;
    Alarm49 : BOOL ;
    Alarm50 : BOOL ;
    Alarm51 : BOOL ;
    Alarm52 : BOOL ;
    Alarm53 : BOOL ;
    Alarm54 : BOOL ;
    Alarm55 : BOOL ;
    Alarm56 : BOOL ;
    Alarm57 : BOOL ;
    Alarm58 : BOOL ;
    Alarm59 : BOOL ;
    Alarm60 : BOOL ;
    Alarm61 : BOOL ;
    Alarm62 : BOOL ;
    Alarm63 : BOOL ;
    Alarm64 : BOOL ;
   END_STRUCT ;
  END_STRUCT ;	
BEGIN
END_DATA_BLOCK

DATA_BLOCK DB 155
VERSION : 0.1
  STRUCT
   Command : STRUCT 	//
    Reset_allarmi : BOOL ;
    TestLampade : BOOL ;
    Abbassa_index_cassetto : BOOL ;
    Alza_index_cassetto : BOOL ;
    Alza_gruppo_piantaggio : BOOL ;
    Abbasa_gruppo_piantaggio : BOOL ;
    Alza_piantaggio : BOOL ;
    Abbasa_piantaggio : BOOL ;
    ris_w2 : DWORD ;
    ris_w6 : DWORD ;
   END_STRUCT ;
   State : STRUCT 	//da indirizzo 10
    Porte_chiuse : BOOL ;
    Porte_chiuse_e_bloccate : BOOL ;
    Cassetto_dentro : BOOL ;
    Cassetto_fuori : BOOL ;
    Index_cassetto_basso : BOOL ;
    Index_cassetto_alto : BOOL ;
    Gruppo_piantaggio_alto : BOOL ;
    Gruppo_piantaggio_basso : BOOL ;
    Piantaggio_alto : BOOL ;
    Piantaggio_basso : BOOL ;
    Piantaggiofinito : BOOL ;
    Piantaggio_pezzo_OK : BOOL ;
    Piantaggio_pezzo_KO : BOOL ;
    FP_Mode_automatic : BOOL ;
    FP_uscita_da_allarme : BOOL ;
    FP_Cassettodentro : BOOL ;
    CassetDentroInizioCiclo : BOOL ;
    ris_w24 : WORD ;
    ris_w6 : DWORD ;
   END_STRUCT ;
   Data : STRUCT 	//da indirizzo 20
    frr1 : BOOL ;
    ris_w2 : DWORD ;
    ris_w6 : DWORD ;
   END_STRUCT ;
  END_STRUCT ;	
BEGIN
   State.Porte_chiuse := TRUE;
   State.Porte_chiuse_e_bloccate := TRUE;
   State.Cassetto_dentro := TRUE;
   State.Index_cassetto_basso := TRUE;
   State.Gruppo_piantaggio_alto := TRUE;
   State.Piantaggio_alto := TRUE;
   State.Piantaggio_pezzo_OK := TRUE;
END_DATA_BLOCK

DATA_BLOCK DB 156
VERSION : 0.1
  STRUCT
   ToolCode_Bit_0 : BOOL ;	//
   ToolCode_Bit_1 : BOOL ;
   ToolCode_Bit_2 : BOOL ;
   ToolCode_Bit_3 : BOOL ;
   ToolCode_Bit_4 : BOOL ;
   Ris_0_05 : BOOL ;
   Ris_0_06 : BOOL ;
   Ris_0_07 : BOOL ;
  END_STRUCT ;	
BEGIN
END_DATA_BLOCK

DATA_BLOCK DB 158
VERSION : 0.1
  STRUCT
   DB_VAR : INT ;	//Variabile jolly provvisoria
  END_STRUCT ;	
BEGIN
END_DATA_BLOCK

DATA_BLOCK DB 160
VERSION : 0.1
  STRUCT
   ID_Ricetta : INT ;
   PartNumber : ARRAY  [0 .. 31 ] OF //Part number in lavorazione
   CHAR ;
   ToolType : INT ;	//Tool type
   ToolCode : INT ;	//Codice su attrezzo - ingressi digitali
   spare38 : DINT ;
   spare42 : DINT ;
   spare46 : DINT ;
   spare50 : ARRAY  [0 .. 13 ] OF INT ;
   Disable : STRUCT 	//da indirizzo 78
    CkCodicePortapezzo : BOOL ;
    CheckSpare50_1 : BOOL ;
    CheckSpare50_2 : BOOL ;
    CheckSpare50_3 : BOOL ;
    CheckSpare50_4 : BOOL ;
    CheckSpare50_5 : BOOL ;
    CheckSpare50_6 : BOOL ;
    CheckSpare50_7 : BOOL ;
    CheckSpare51_0 : BOOL ;
    CheckSpare51_1 : BOOL ;
   END_STRUCT ;
   Corsa_piantaggio_min : REAL ;	//mm
   Corsa_piantaggio_max : REAL ;	//mm
   Spare_88 : REAL ;	//
   Tempo_stabilizzazione : DINT ;	//Millisecondi
   Timeout_piantaggio : DINT ;	//millisecondi
   spare100 : INT ;
   spare102 : INT ;
   spare104 : INT ;
   spare106 : INT ;
   spare108 : INT ;
   spare110 : ARRAY  [0 .. 145 ] OF INT ;
  END_STRUCT ;	
BEGIN
   ID_Ricetta := 1;
   PartNumber[0] := 'R';
   PartNumber[1] := 'P';
   PartNumber[2] := 'V';
   PartNumber[3] := 'O';
   PartNumber[4] := ' ';
   PartNumber[5] := 'A';
   PartNumber[6] := 'P';
   PartNumber[7] := 'O';
   PartNumber[8] := '0';
   PartNumber[9] := '2';
   PartNumber[10] := ' ';
   PartNumber[11] := ' ';
   PartNumber[12] := ' ';
   PartNumber[13] := ' ';
   PartNumber[14] := ' ';
   PartNumber[15] := ' ';
   PartNumber[16] := ' ';
   PartNumber[17] := ' ';
   PartNumber[18] := ' ';
   PartNumber[19] := ' ';
   PartNumber[20] := ' ';
   PartNumber[21] := ' ';
   PartNumber[22] := ' ';
   PartNumber[23] := ' ';
   PartNumber[24] := ' ';
   PartNumber[25] := ' ';
   PartNumber[26] := ' ';
   PartNumber[27] := ' ';
   PartNumber[28] := ' ';
   PartNumber[29] := ' ';
   PartNumber[30] := ' ';
   PartNumber[31] := ' ';
   ToolType := 1;
   ToolCode := 1;
   Corsa_piantaggio_min := 2.000000e-01;
   Corsa_piantaggio_max := 8.000000e-01;
   Spare_88 := 5.000000e+00;
   Tempo_stabilizzazione := L#3000;
   Timeout_piantaggio := L#10000;
END_DATA_BLOCK

DATA_BLOCK DB 170
VERSION : 0.1
  STRUCT
   General : UDT 200;
   Restore : UDT 200;
  END_STRUCT ;	
BEGIN
// 44 bytes; values not shown
END_DATA_BLOCK

DATA_BLOCK DB 200
VERSION : 0.1
UDT 250
BEGIN
END_DATA_BLOCK

DATA_BLOCK DB 201
VERSION : 0.1
  STRUCT
   P_Consenso_operatore : BOOL ;	//(start ciclo)
   Pipe_posizionato : BOOL ;
   Cassetto_fuori : BOOL ;
   Cassetto_dentro : BOOL ;
   Index_cassetto_Giu : BOOL ;
   Index_cassetto_Su : BOOL ;
   Sblocco_pezzo_Giu : BOOL ;
   Sblocco_pezzo_Su : BOOL ;
   PulStopCiclo : BOOL ;
  END_STRUCT ;	
BEGIN
   Cassetto_fuori := TRUE;
   Index_cassetto_Su := TRUE;
   Sblocco_pezzo_Su := TRUE;
END_DATA_BLOCK

DATA_BLOCK DB 202
VERSION : 0.1
  STRUCT
   Fine_ciclo_OK : BOOL ;	//
   Fine_ciclo_NON_OK : BOOL ;
   EV_abb_index_cassetto : BOOL ;	//Libera index cassetto su zona piantaggio
   EV_alza_index_cassetto : BOOL ;	//Blocca index cassetto su zona piantaggio
   EV_sblocco_pezzo : BOOL ;
   EV_blocco_pezzo : BOOL ;
  END_STRUCT ;	
BEGIN
   EV_alza_index_cassetto := TRUE;
   EV_sblocco_pezzo := TRUE;
END_DATA_BLOCK

DATA_BLOCK DB 203
VERSION : 0.1
  STRUCT
   Dummy : INT ;	//
  END_STRUCT ;	
BEGIN
END_DATA_BLOCK

DATA_BLOCK DB 204
VERSION : 0.1
  STRUCT
   Emegency : STRUCT
    Alarm01 : BOOL ;	//OP40 ToolType error
    Alarm02 : BOOL ;	//OP40 Tool Code error
    Alarm03 : BOOL ;
    Alarm04 : BOOL ;
    Alarm05 : BOOL ;
    Alarm06 : BOOL ;
    Alarm07 : BOOL ;
    Alarm08 : BOOL ;
    Alarm09 : BOOL ;	//
    Alarm10 : BOOL ;	//
    Alarm11 : BOOL ;	//
    Alarm12 : BOOL ;	//
    Alarm13 : BOOL ;	//
    Alarm14 : BOOL ;	//
    Alarm15 : BOOL ;
    Alarm16 : BOOL ;
    Alarm17 : BOOL ;
    Alarm18 : BOOL ;
    Alarm19 : BOOL ;
    Alarm20 : BOOL ;
    Alarm21 : BOOL ;
    Alarm22 : BOOL ;
    Alarm23 : BOOL ;
    Alarm24 : BOOL ;
    Alarm25 : BOOL ;
    Alarm26 : BOOL ;
    Alarm27 : BOOL ;
    Alarm28 : BOOL ;
    Alarm29 : BOOL ;
    Alarm30 : BOOL ;
    Alarm31 : BOOL ;
    Alarm32 : BOOL ;
    Alarm33 : BOOL ;
    Alarm34 : BOOL ;
    Alarm35 : BOOL ;
    Alarm36 : BOOL ;
    Alarm37 : BOOL ;
    Alarm38 : BOOL ;
    Alarm39 : BOOL ;
    Alarm40 : BOOL ;
    Alarm41 : BOOL ;
    Alarm42 : BOOL ;
    Alarm43 : BOOL ;
    Alarm44 : BOOL ;
    Alarm45 : BOOL ;
    Alarm46 : BOOL ;
    Alarm47 : BOOL ;
    Alarm48 : BOOL ;
    Alarm49 : BOOL ;
    Alarm50 : BOOL ;
    Alarm51 : BOOL ;
    Alarm52 : BOOL ;
    Alarm53 : BOOL ;
    Alarm54 : BOOL ;
    Alarm55 : BOOL ;
    Alarm56 : BOOL ;
    Alarm57 : BOOL ;
    Alarm58 : BOOL ;
    Alarm59 : BOOL ;
    Alarm60 : BOOL ;
    Alarm61 : BOOL ;
    Alarm62 : BOOL ;
    Alarm63 : BOOL ;
    Alarm64 : BOOL ;
   END_STRUCT ;
   StopCycle : STRUCT
    Alarm01 : BOOL ;	//Errore rilevamento anello di adattamento 1
    Alarm02 : BOOL ;	//Errore rilevamento anello di adattamento 2
    Alarm03 : BOOL ;	//Index cassetto non alto
    Alarm04 : BOOL ;	//Index cassetto non basso
    Alarm05 : BOOL ;	//Incongruenza sensori index cassetto
    Alarm06 : BOOL ;	//Cilindro sblocco pezzo non avanti
    Alarm07 : BOOL ;	//Cilindro sblocco pezzo non indietro
    Alarm08 : BOOL ;	//Incongruenza sensori cilindro sblocco pezzo
    Alarm09 : BOOL ;	//OP40 ToolType error
    Alarm10 : BOOL ;	//OP40 Tool Code error
    Alarm11 : BOOL ;
    Alarm12 : BOOL ;
    Alarm13 : BOOL ;
    Alarm14 : BOOL ;
    Alarm15 : BOOL ;
    Alarm16 : BOOL ;
    Alarm17 : BOOL ;
    Alarm18 : BOOL ;
    Alarm19 : BOOL ;
    Alarm20 : BOOL ;
    Alarm21 : BOOL ;
    Alarm22 : BOOL ;
    Alarm23 : BOOL ;
    Alarm24 : BOOL ;
    Alarm25 : BOOL ;
    Alarm26 : BOOL ;
    Alarm27 : BOOL ;
    Alarm28 : BOOL ;
    Alarm29 : BOOL ;
    Alarm30 : BOOL ;
    Alarm31 : BOOL ;
    Alarm32 : BOOL ;
    Alarm33 : BOOL ;
    Alarm34 : BOOL ;
    Alarm35 : BOOL ;
    Alarm36 : BOOL ;
    Alarm37 : BOOL ;
    Alarm38 : BOOL ;
    Alarm39 : BOOL ;
    Alarm40 : BOOL ;
    Alarm41 : BOOL ;
    Alarm42 : BOOL ;
    Alarm43 : BOOL ;
    Alarm44 : BOOL ;
    Alarm45 : BOOL ;
    Alarm46 : BOOL ;
    Alarm47 : BOOL ;
    Alarm48 : BOOL ;
    Alarm49 : BOOL ;
    Alarm50 : BOOL ;
    Alarm51 : BOOL ;
    Alarm52 : BOOL ;
    Alarm53 : BOOL ;
    Alarm54 : BOOL ;
    Alarm55 : BOOL ;
    Alarm56 : BOOL ;
    Alarm57 : BOOL ;
    Alarm58 : BOOL ;
    Alarm59 : BOOL ;
    Alarm60 : BOOL ;
    Alarm61 : BOOL ;
    Alarm62 : BOOL ;
    Alarm63 : BOOL ;
    Alarm64 : BOOL ;
   END_STRUCT ;
   RestartCycle : STRUCT
    Alarm01 : BOOL ;
    Alarm02 : BOOL ;
    Alarm03 : BOOL ;
    Alarm04 : BOOL ;
    Alarm05 : BOOL ;
    Alarm06 : BOOL ;
    Alarm07 : BOOL ;
    Alarm08 : BOOL ;
    Alarm09 : BOOL ;
    Alarm10 : BOOL ;
    Alarm11 : BOOL ;
    Alarm12 : BOOL ;
    Alarm13 : BOOL ;
    Alarm14 : BOOL ;
    Alarm15 : BOOL ;
    Alarm16 : BOOL ;
    Alarm17 : BOOL ;
    Alarm18 : BOOL ;
    Alarm19 : BOOL ;
    Alarm20 : BOOL ;
    Alarm21 : BOOL ;
    Alarm22 : BOOL ;
    Alarm23 : BOOL ;
    Alarm24 : BOOL ;
    Alarm25 : BOOL ;
    Alarm26 : BOOL ;
    Alarm27 : BOOL ;
    Alarm28 : BOOL ;
    Alarm29 : BOOL ;
    Alarm30 : BOOL ;
    Alarm31 : BOOL ;
    Alarm32 : BOOL ;
    Alarm33 : BOOL ;
    Alarm34 : BOOL ;
    Alarm35 : BOOL ;
    Alarm36 : BOOL ;
    Alarm37 : BOOL ;
    Alarm38 : BOOL ;
    Alarm39 : BOOL ;
    Alarm40 : BOOL ;
    Alarm41 : BOOL ;
    Alarm42 : BOOL ;
    Alarm43 : BOOL ;
    Alarm44 : BOOL ;
    Alarm45 : BOOL ;
    Alarm46 : BOOL ;
    Alarm47 : BOOL ;
    Alarm48 : BOOL ;
    Alarm49 : BOOL ;
    Alarm50 : BOOL ;
    Alarm51 : BOOL ;
    Alarm52 : BOOL ;
    Alarm53 : BOOL ;
    Alarm54 : BOOL ;
    Alarm55 : BOOL ;
    Alarm56 : BOOL ;
    Alarm57 : BOOL ;
    Alarm58 : BOOL ;
    Alarm59 : BOOL ;
    Alarm60 : BOOL ;
    Alarm61 : BOOL ;
    Alarm62 : BOOL ;
    Alarm63 : BOOL ;
    Alarm64 : BOOL ;
   END_STRUCT ;
   Warning : STRUCT
    Alarm01 : BOOL ;	//Blocco movimento index cassetto se cassetto non dentro o non fuori
    Alarm02 : BOOL ;	//Blocco sblocco pezzo se cassetto non fuori
    Alarm03 : BOOL ;	//Sblocco index solo con ribaditrice alta
    Alarm04 : BOOL ;	//Sblocco index solo con assi fermi
    Alarm05 : BOOL ;	//Sblocco index solo pezzo bloccato
    Alarm06 : BOOL ;
    Alarm07 : BOOL ;
    Alarm08 : BOOL ;
    Alarm09 : BOOL ;
    Alarm10 : BOOL ;
    Alarm11 : BOOL ;
    Alarm12 : BOOL ;
    Alarm13 : BOOL ;
    Alarm14 : BOOL ;
    Alarm15 : BOOL ;
    Alarm16 : BOOL ;
    Alarm17 : BOOL ;
    Alarm18 : BOOL ;
    Alarm19 : BOOL ;
    Alarm20 : BOOL ;
    Alarm21 : BOOL ;
    Alarm22 : BOOL ;
    Alarm23 : BOOL ;
    Alarm24 : BOOL ;
    Alarm25 : BOOL ;
    Alarm26 : BOOL ;
    Alarm27 : BOOL ;
    Alarm28 : BOOL ;
    Alarm29 : BOOL ;
    Alarm30 : BOOL ;
    Alarm31 : BOOL ;
    Alarm32 : BOOL ;
    Alarm33 : BOOL ;
    Alarm34 : BOOL ;
    Alarm35 : BOOL ;
    Alarm36 : BOOL ;
    Alarm37 : BOOL ;
    Alarm38 : BOOL ;
    Alarm39 : BOOL ;
    Alarm40 : BOOL ;
    Alarm41 : BOOL ;
    Alarm42 : BOOL ;
    Alarm43 : BOOL ;
    Alarm44 : BOOL ;
    Alarm45 : BOOL ;
    Alarm46 : BOOL ;
    Alarm47 : BOOL ;
    Alarm48 : BOOL ;
    Alarm49 : BOOL ;
    Alarm50 : BOOL ;
    Alarm51 : BOOL ;
    Alarm52 : BOOL ;
    Alarm53 : BOOL ;
    Alarm54 : BOOL ;
    Alarm55 : BOOL ;
    Alarm56 : BOOL ;
    Alarm57 : BOOL ;
    Alarm58 : BOOL ;
    Alarm59 : BOOL ;
    Alarm60 : BOOL ;
    Alarm61 : BOOL ;
    Alarm62 : BOOL ;
    Alarm63 : BOOL ;
    Alarm64 : BOOL ;
   END_STRUCT ;
  END_STRUCT ;	
BEGIN
END_DATA_BLOCK

DATA_BLOCK DB 205
VERSION : 0.1
  STRUCT
   Command : STRUCT 	//
    Reset_allarmi : BOOL ;
    TestLampade : BOOL ;
    Abbassa_index_cassetto : BOOL ;
    Alza_index_cassetto : BOOL ;
    Sblocca_pezzo : BOOL ;
    Blocca_pezzo : BOOL ;
    FP_Consenso_operatore : BOOL ;
    Prenota_ribaditrice : BOOL ;
    Vai_in_posizione_assi : BOOL ;
    Marcia_ribaditrice : BOOL ;
    Abbassa_ribaditrice : BOOL ;
    Alza_ribaditrice : BOOL ;
    ris_w2 : DWORD ;
    ris_w6 : DWORD ;
   END_STRUCT ;
   State : STRUCT 	//da indirizzo 10
    Porte_chiuse : BOOL ;
    Porte_chiuse_e_bloccate : BOOL ;
    Cassetto_dentro : BOOL ;
    Cassetto_fuori : BOOL ;
    Index_cassetto_basso : BOOL ;
    Index_cassetto_alto : BOOL ;
    Pezzo_sbloccato : BOOL ;
    Pezzo_bloccato : BOOL ;
    _Ribaditrice_a_disposiz : BOOL ;
    _Assi_posiz_raggiunta : BOOL ;
    Ribaditura_effettuata : BOOL ;
    Ribaditrice_alta : BOOL ;
    Ribaditrice_bassa : BOOL ;
    Ribaditrice_in_marcia : BOOL ;
    FP_stato_20_generale : BOOL ;
    _Ribad_in_fuori_ingombro : BOOL ;
    FP_Mode_automatic : BOOL ;
    FP_uscita_da_allarme : BOOL ;
    Ribaditura_pezzo_OK : BOOL ;
    Ribaditura_pezzo_KO : BOOL ;
    Assi_fermi : BOOL ;
    ris_w4 : WORD ;
    ris_w6 : DWORD ;
   END_STRUCT ;
   Data : STRUCT 	//da indirizzo 20
    Num_punto_in_lavorazione : INT ;
    Pos_comandata_asse_X : DINT ;	//Punto in lavorazione
    Pos_comandata_asse_Y : DINT ;	//Punto in lavorazione
    Tempo_ribaditura : DINT ;	//Punto in lavorazione
    ris_w2 : DWORD ;
    ris_w6 : DWORD ;
   END_STRUCT ;
  END_STRUCT ;	
BEGIN
   Command.Sblocca_pezzo := TRUE;
   State.Porte_chiuse := TRUE;
   State.Porte_chiuse_e_bloccate := TRUE;
   State.Cassetto_fuori := TRUE;
   State.Index_cassetto_alto := TRUE;
   State.Pezzo_sbloccato := TRUE;
   State.Ribaditrice_alta := TRUE;
   State.Assi_fermi := TRUE;
END_DATA_BLOCK

DATA_BLOCK DB 206
VERSION : 0.1
  STRUCT
   ToolCode_Bit_0 : BOOL ;	//
   ToolCode_Bit_1 : BOOL ;
   ToolCode_Bit_2 : BOOL ;
   ToolCode_Bit_3 : BOOL ;
   ToolCode_Bit_4 : BOOL ;
   Anello_1_Inserito : BOOL ;
   Anello_2_Inserito : BOOL ;
   Presenza_nozzle_ring : BOOL ;
  END_STRUCT ;	
BEGIN
   ToolCode_Bit_0 := TRUE;
   ToolCode_Bit_1 := TRUE;
   Anello_2_Inserito := TRUE;
END_DATA_BLOCK

DATA_BLOCK DB 208
VERSION : 0.1
  STRUCT
   DB_VAR : INT ;	//Variabile jolly provvisoria
  END_STRUCT ;	
BEGIN
END_DATA_BLOCK

DATA_BLOCK DB 209
VERSION : 0.1
  STRUCT
   DB_VAR : INT ;	//Variabile jolly provvisoria
  END_STRUCT ;	
BEGIN
END_DATA_BLOCK

